# B&R Automation Studio project Kesim (part 3)

#### Park.st
```iecst
ACTION Park:

	CASE gMain.Out.MainSubStep OF

		SUB_INIT:

			IF Loc.FirstInSubState THEN
				gAxBasic[AX_X].MoveAbsolute		:= FALSE;
				gAxBasic[AX_Y].MoveAbsolute		:= FALSE;
				gAxBasic[AX_C].MoveAbsolute		:= FALSE;
				gIO.Out.CT.CuttingHeadDown 		:= FALSE;
				gIO.Out.CT.LowEMotorDown   		:= FALSE;
				gIO.Out.CT.FanStart		   		:= FALSE;
				gIO.Out.CT.XYGlassBreakControl  := FALSE;
				gIO.Out.CT.TransferBelt			:= FALSE;
				gIO.Out.CT.SquareForward		:= FALSE;
			ELSE
				Loc.Timers.TON_ParkState.IN := TRUE;
				Loc.Timers.TON_ParkState.PT := T#1s;
				IF Loc.Timers.TON_ParkState.Q THEN
					Loc.Timers.TON_ParkState.IN := FALSE;
					gMain.Out.MainSubStep			:= PARK_CHECK_IO;
				END_IF
			END_IF;

		PARK_CHECK_IO:
			IF NOT gIO.In.CT.HeadMaxDownSensor THEN
				gMain.Out.Error 	:= TRUE;
				gMain.Out.ErrorID 	:= 999; // Diamond Is Not Back
				gMain.Out.MainSubStep   	:= SUB_ERROR;
				RETURN;

			ELSIF gParameters.MachineType = OCKM THEN
				IF NOT gIO.In.CT.TableDownStopSwicth OR gIO.In.CT.TableUpSlowSwicth ELSE
					gMain.Out.Error 	:= TRUE;
					gMain.Out.ErrorID 	:= 999; // CT_Is_Not_Down
					gMain.Out.MainSubStep   	:= PARK_ERROR;
					RETURN;
					ELSIF NOT gIO.In.CT.TableSquareBack THEN
					gMain.Out.Error 	:= TRUE;
					gMain.Out.ErrorID 	:= 999; // CT_Is_Squares_Are_Not_Back
					gMain.Out.MainSubStep   	:= PARK_ERROR;
					RETURN;
				ELSE
					gMain.Out.MainSubStep   	:= SUB_PARK_START;
				END_IF // OCKM
			ELSIF gParameters.MachineType = FCL THEN
				IF NOT gIO.In.CT.GlassTransBeltIsDown ELSE
					gMain.Out.Error 	:= TRUE;
					gMain.Out.ErrorID 	:= 999; // CT_Belt Is Not Down
					gMain.Out.MainSubStep   	:= SUB_ERROR;
					RETURN;
				END_IF // FCL
			ELSE
				gMain.Out.MainSubStep := SUB_PARK_START;
			END_IF;

			SUB_PARK_START:
				IF Loc.FirstInSubState THEN

					// X Axis Go Park
					gAxBasicPar[AX_X].Acceleration	:= 200.0;
					gAxBasicPar[AX_X].Deceleration 	:= 200.0;
					gAxBasicPar[AX_X].Velocity		:= (gParameters.LengthParametes.ParkSpeed / 100) * C_MAX_CUT_SPEED * (1000/60);
					gAxBasicPar[AX_X].Position 		:= gMain.In.Settings.ParkPos[AX_X];
					gAxBasic[AX_X].MoveAbsolute		:= TRUE;

					// Y Axis Go Park
					gAxBasicPar[AX_Y].Acceleration	:= 200.0;
					gAxBasicPar[AX_Y].Deceleration 	:= 200.0;
					gAxBasicPar[AX_Y].Velocity		:= (gParameters.LengthParametes.ParkSpeed / 100) * C_MAX_CUT_SPEED * (1000/60);
					gAxBasicPar[AX_Y].Position 		:= gMain.In.Settings.ParkPos[AX_Y];
					gAxBasic[AX_Y].MoveAbsolute		:= TRUE;

					// C Axis Go Park
					gAxBasicPar[AX_C].Acceleration	:= 200.0;
					gAxBasicPar[AX_C].Deceleration 	:= 200.0;
					gAxBasicPar[AX_C].Velocity		:= 200.0;
					gAxBasicPar[AX_C].Position 		:= gMain.In.Settings.ParkPos[AX_C];
					gAxBasic[AX_C].MoveAbsolute		:= TRUE;

				ELSE
					IF gAxBasic[AX_X].MoveDone AND gAxBasic[AX_Y].MoveDone AND gAxBasic[AX_C].MoveDone THEN
						gMain.Out.MainSubStep			:= PARK_DONE;
					END_IF;
				END_IF;

			SUB_CMD_DONE:
				IF gMain.Out.Status.Ax_Parked  THEN
					Loc.HomeState			:= SUB_INIT;
					//		gMain.Out.MainStep		:= MAIN_WAIT_CMD;
				END_IF;

			SUB_STOP:

			SUB_ERROR:
			IF Loc.FirstInSubState THEN
				gAxBasic[AX_X].MoveAbsolute		:= FALSE;
				gAxBasic[AX_Y].MoveAbsolute		:= FALSE;
				gAxBasic[AX_C].MoveAbsolute		:= FALSE;
				Loc.Timers.TON_ParkState.IN		:= FALSE;
			ELSE
				IF gMain.In.Cmd.Reset THEN
					gAxBasic[AX_X].ErrorReset		:= TRUE;
					gAxBasic[AX_Y].ErrorReset		:= TRUE;
					gAxBasic[AX_C].ErrorReset		:= TRUE;
				ELSE
					gAxBasic[AX_X].ErrorReset		:= FALSE;
					gAxBasic[AX_Y].ErrorReset		:= FALSE;
					gAxBasic[AX_C].ErrorReset		:= FALSE;
				END_IF;

				IF NOT gAxBasic[ AX_X].Error AND NOT gAxBasic[ AX_Y].Error NOT gAxBasic[ AX_C].Error THEN
					gMain.Out.MainSubStep			:= SUB_INIT;
					//gMain.Out.MainStep		:= MAIN_WAIT_CMD;
				END_IF;

			END_IF;

		END_CASE;

		Loc.Timers.TON_ParkState();

		END_ACTION
```

### Program Logical/SourceCode/CncCtrl (IEC)

#### Main.st - Init, cyclic, exit code
```iecst
(********************************************************************
 * COPYRIGHT --  B&R Industrial Automation GmbH
 ********************************************************************
 * Task: SUB0
 * Author: kay3a
 * Created: October 16, 2024/11:06 AM
 ********************************************************************
 * Description: Machine CncCtrl task
 ********************************************************************)
PROGRAM _INIT

	//|ŻŻŻŻŻŻŻŻŻŻŻŻŻŻŻŻŻŻŻŻŻŻŻŻŻŻŻŻŻŻŻŻŻŻŻŻŻŻŻŻŻŻŻŻŻŻŻŻŻŻŻŻŻŻŻŻŻŻŻŻŻŻŻŻŻŻŻŻŻŻŻŻŻ
	//|               CNC Klasörünü olustur
	//|_________________________________________________________________________
	Loc.FB.DirCreate.Parameters.DeviceName := 'DEV_CNC';
	Loc.FB.DirCreate.Parameters.DirPath := '/DEVICE=USER_PATH/CNC';
	Loc.FB.DirCreate.Enable := TRUE;
	REPEAT
		Loc.FB.DirCreate.Execute := Loc.FB.DirCreate.Active AND NOT Loc.FB.DirCreate.CommandBusy AND NOT Loc.FB.DirCreate.CommandDone;
		Loc.FB.DirCreate();
		UNTIL Loc.FB.DirCreate.CommandDone
	END_REPEAT;
	//|_________________________________________________________________________

	//|ŻŻŻŻŻŻŻŻŻŻŻŻŻŻŻŻŻŻŻŻŻŻŻŻŻŻŻŻŻŻŻŻŻŻŻŻŻŻŻŻŻŻŻŻŻŻŻŻŻŻŻŻŻŻŻŻŻŻŻŻŻŻŻŻŻŻŻŻŻŻŻŻŻ
	//|               CNC File olustur
	//|_________________________________________________________________________
	Loc.FB.FileCreate.Parameters.DeviceName := 'DEV_CNC';
	Loc.FB.FileCreate.Parameters.FileName := 'Program.cnc';
	Loc.FB.FileCreate.Enable := TRUE;
	REPEAT
		Loc.FB.FileCreate.Execute := Loc.FB.FileCreate.Active AND NOT Loc.FB.FileCreate.CommandBusy AND NOT Loc.FB.FileCreate.CommandDone;
		Loc.FB.FileCreate();
		UNTIL Loc.FB.FileCreate.CommandDone
	END_REPEAT;
	//|_________________________________________________________________________

	//|ŻŻŻŻŻŻŻŻŻŻŻŻŻŻŻŻŻŻŻŻŻŻŻŻŻŻŻŻŻŻŻŻŻŻŻŻŻŻŻŻŻŻŻŻŻŻŻŻŻŻŻŻŻŻŻŻŻŻŻŻŻŻŻŻŻŻŻŻŻŻŻŻŻ
	//|               L I V E    F B s
	//|_________________________________________________________________________
//	(* PML *)
//	Loc.FB.PML.MpLink := ADR(gMpLink_PackMLSyncModule_CncCtrl);
//	Loc.FB.PML.Parameters := ADR(Loc.Par.PML);
//	Loc.FB.PML.Enable := TRUE;

	(* CNC *)
	Loc.FB.Cnc3Axis.MpLink := ADR(gMpLink_CncXYZ);
	Loc.FB.Cnc3Axis.Parameters := ADR(Loc.Par.Cnc3Axis);
	Loc.FB.Cnc3Axis.Enable := TRUE;
	Loc.FB.Cnc3Axis.Override := 100.0;
	// Par
	Loc.Par.Cnc3Axis.ProgramName := 'Program.cnc';
	//|_________________________________________________________________________

END_PROGRAM

PROGRAM _CYCLIC

	(* Axis *)
	Loc.FB.Cnc3Axis();

	//|_________________________________________________________________________
	TestX := Loc.FB.Cnc3Axis.X / 1500;
	TestY := Loc.FB.Cnc3Axis.Z / 1500;

  gCncAdress := ADR ( Loc.FB.Cnc3Axis );

END_PROGRAM

PROGRAM _EXIT

	//|ŻŻŻŻŻŻŻŻŻŻŻŻŻŻŻŻŻŻŻŻŻŻŻŻŻŻŻŻŻŻŻŻŻŻŻŻŻŻŻŻŻŻŻŻŻŻŻŻŻŻŻŻŻŻŻŻŻŻŻŻŻŻŻŻŻŻŻŻŻŻŻŻŻ
	//|              K I L L   F B s
	//|_________________________________________________________________________
	(* PML *)
//	Loc.FB.PML(Enable := FALSE);

	(* CNC *)
	Loc.FB.Cnc3Axis(Enable := FALSE);
	//|_________________________________________________________________________

END_PROGRAM
```

#### Types.typ - Local data types
```iecst
(********************************************************************
 * COPYRIGHT --  B&R Industrial Automation GmbH
 *******************************************************************
 * Task: MAIN
 * Author: kay3a
 * Created: October 16, 2024/11:08 AM
 ********************************************************************)

TYPE
	Loc_typ : 	STRUCT  (**** Local Type*)
		FB : Loc_FB_typ; (**** Local FB Type*)
		Par : Loc_Par_typ;
		Cmd : Loc_Cmd_typ; (**** Local Command Type*)
		Status : Loc_Status_typ; (**** Local Status Type*)
	END_STRUCT;
END_TYPE

(**)
(**** Local FB Type*)

TYPE
	Loc_FB_typ : 	STRUCT  (**** Local FB Type*)
		Cnc3Axis : MpCnc3Axis; (**** CNC FB*)
		DirCreate : FbDirCreate; (**** CNC Direction create*)
		FileCreate : FbFileCreate; (**** CNC File create*)
	END_STRUCT;
END_TYPE

(**)
(**** Local Par Type*)

TYPE
	Loc_Par_typ : 	STRUCT  (**** Local Par Type*)
		Cnc3Axis : MpCnc3AxisParType;
	END_STRUCT;
END_TYPE

(**)
(**** Local Cmd Type*)

TYPE
	Loc_Cmd_typ : 	STRUCT  (**** Local Cmd Type*)
		New_Member : USINT;
	END_STRUCT;
END_TYPE

(**)
(**** Local Status Type*)

TYPE
	Loc_Status_typ : 	STRUCT  (**** Local Status Type*)
		New_Member : USINT;
	END_STRUCT;
END_TYPE

(**)
```

#### Variables.var - Local variables
```iecst
(********************************************************************
 * COPYRIGHT --  B&R Industrial Automation GmbH
 *******************************************************************
 * Task: MAIN
 * Author: kay3a
 * Created: October 16, 2024/11:08 AM
 ********************************************************************)
VAR
	Loc : Loc_typ; (**** Bu Task icinde kullanilacak Local degisken*)
	TestY : LREAL;
	TestX : LREAL;
END_VAR
```

#### Package Logical/SourceCode/CncCtrl/act_PML - PackML specific actions are stored in this package.

#### Execute.st
```iecst
(*********************************************************************************
 * Copyright: B&R Industrial Automation GmbH
 * Author:    kay3a
 * Created:   June 21, 2023/5:55 PM
 *********************************************************************************)
ACTION Execute:

END_ACTION

ACTION Execute_Manual:

END_ACTION

ACTION Execute_Production:

END_ACTION
```

#### Starting.st
```iecst
(*********************************************************************************
 * Copyright: B&R Industrial Automation GmbH
 * Author:    kay3a
 * Created:   June 21, 2023/5:55 PM
 *********************************************************************************)
ACTION Starting:

	Loc.FB.PML.Command.StateComplete := TRUE;

END_ACTION
```

#### Stopping.st
```iecst
(*********************************************************************************
 * Copyright: B&R Industrial Automation GmbH
 * Author:    kay3a
 * Created:   June 21, 2023/5:55 PM
 *********************************************************************************)
ACTION Stopping:

Loc.FB.PML.Command.StateComplete := TRUE;

END_ACTION
```

#### Completing.st
```iecst
(*********************************************************************************
 * Copyright: B&R Industrial Automation GmbH
 * Author:    kay3a
 * Created:   June 21, 2023/5:55 PM
 *********************************************************************************)
ACTION Completing:

Loc.FB.PML.Command.StateComplete := TRUE;

END_ACTION
```

#### Suspended.st
```iecst
(*********************************************************************************
 * Copyright: B&R Industrial Automation GmbH
 * Author:    kay3a
 * Created:   June 21, 2023/5:55 PM
 *********************************************************************************)
ACTION Suspended:

Loc.FB.PML.Command.StateComplete := TRUE;

END_ACTION
```

#### Complete.st
```iecst
(*********************************************************************************
 * Copyright: B&R Industrial Automation GmbH
 * Author:    kay3a
 * Created:   June 21, 2023/5:55 PM
 *********************************************************************************)
ACTION Complete:

END_ACTION
```

#### Idle.st
```iecst
(*********************************************************************************
 * Copyright: B&R Industrial Automation GmbH
 * Author:    kay3a
 * Created:   June 21, 2023/5:55 PM
 *********************************************************************************)
ACTION Idle:

END_ACTION
```

#### Unholding.st
```iecst
(*********************************************************************************
 * Copyright: B&R Industrial Automation GmbH
 * Author:    kay3a
 * Created:   June 21, 2023/5:55 PM
 *********************************************************************************)
ACTION Unholding:

	Loc.FB.PML.Command.StateComplete := TRUE;

END_ACTION
```

#### Held.st
```iecst
(*********************************************************************************
 * Copyright: B&R Industrial Automation GmbH
 * Author:    kay3a
 * Created:   June 21, 2023/5:55 PM
 *********************************************************************************)
ACTION Held:

END_ACTION
```

- sample.pptx (binary file, 35832 bytes)
#### GCode_Ref.txt
```
%001 (CncProgram)

N10 G90     (absolute coordinates)
N20 F10000    (Feed rate in measurements units/min)

(* Glass Height:1500mm
(* Glass Length:1000mm  *)

G04 3
G01 X 0  Y0  Z0
G01 X-1000
G01 Y-90
G01 Z1000

G03  G18 I500 H180   Z1000 Y-270

G01 Z0
```

### Program Logical/SourceCode/Infastructure/AlarmX (IEC)

#### Main.st - Init, cyclic, exit code
```iecst
(********************************************************************
 * COPYRIGHT --  B&R Industrial Automation GmbH
 ********************************************************************
 * Task: AlarmX
 * Author: kay3a
 * Created: October 2, 2024/3:55 PM
 ********************************************************************
 * Description: Alarm mgr
 ********************************************************************)
PROGRAM _INIT

	//|ŻŻŻŻŻŻŻŻŻŻŻŻŻŻŻŻŻŻŻŻŻŻŻŻŻŻŻŻŻŻŻŻŻŻŻŻŻŻŻŻŻŻŻŻŻŻŻŻŻŻŻŻŻŻŻŻŻŻŻŻŻŻŻŻŻŻŻŻŻŻŻŻŻ
	//|               AlarmXHistory Klasörünü olustur
	//|_________________________________________________________________________
	Loc.FB.DirCreate.Parameters.DeviceName := 'DEV_ALARM';
	Loc.FB.DirCreate.Parameters.DirPath := '/DEVICE=USER_PATH/AlarmX';
	Loc.FB.DirCreate.Enable := TRUE;
	REPEAT
		Loc.FB.DirCreate.Execute := Loc.FB.DirCreate.Active AND NOT Loc.FB.DirCreate.CommandBusy AND NOT Loc.FB.DirCreate.CommandDone;
		Loc.FB.DirCreate();
		UNTIL Loc.FB.DirCreate.CommandDone
	END_REPEAT;
	//|_________________________________________________________________________

	//|ŻŻŻŻŻŻŻŻŻŻŻŻŻŻŻŻŻŻŻŻŻŻŻŻŻŻŻŻŻŻŻŻŻŻŻŻŻŻŻŻŻŻŻŻŻŻŻŻŻŻŻŻŻŻŻŻŻŻŻŻŻŻŻŻŻŻŻŻŻŻŻŻŻ
	//|               FB linklemeleri
	//|_________________________________________________________________________
	(* AlarmXCore *)
	Loc.FB.AlarmXCore.MpLink := ADR(gMpLink_AlarmXCore);
	Loc.FB.AlarmXCore.Enable := TRUE;
	Loc.FB.AlarmXCore();

	(* AlarmXHistory *)
	Loc.FB.AlarmXHistory.Enable := TRUE;
	Loc.FB.AlarmXHistory.MpLink := ADR(gMpLink_AlarmXHistory);
	Loc.FB.AlarmXHistory.FileName := ADR('Alarms_%Y_%m_%d_%H_%M_%S');
	Loc.FB.AlarmXHistory.DeviceName := ADR('DEV_ALARM');
	Loc.FB.AlarmXHistory();
	//|_________________________________________________________________________

	//|ŻŻŻŻŻŻŻŻŻŻŻŻŻŻŻŻŻŻŻŻŻŻŻŻŻŻŻŻŻŻŻŻŻŻŻŻŻŻŻŻŻŻŻŻŻŻŻŻŻŻŻŻŻŻŻŻŻŻŻŻŻŻŻŻŻŻŻŻŻŻŻŻŻ
	//|               Ilk Açilis AlarmHist temizle
	//|_________________________________________________________________________
//	Loc.FB.AlarmXHistory.Clear := TRUE; // bc25.10.15
	//|_________________________________________________________________________

END_PROGRAM

PROGRAM _CYCLIC

	//|ŻŻŻŻŻŻŻŻŻŻŻŻŻŻŻŻŻŻŻŻŻŻŻŻŻŻŻŻŻŻŻŻŻŻŻŻŻŻŻŻŻŻŻŻŻŻŻŻŻŻŻŻŻŻŻŻŻŻŻŻŻŻŻŻŻŻŻŻŻŻŻŻŻ
	//|                Command set/reset
	//|_________________________________________________________________________
	(* AlarmXHistory FB --- ErrorReset *)
	IF Loc.FB.AlarmXHistory.Error THEN
		Loc.FB.AlarmXHistory.ErrorReset := TRUE;
	ELSE
		Loc.FB.AlarmXHistory.ErrorReset := FALSE;
	END_IF;

	(* AlarmXCore FB --- ErrorReset *)
	IF Loc.FB.AlarmXCore.Error THEN
		Loc.FB.AlarmXCore.ErrorReset := TRUE;
	ELSE
		Loc.FB.AlarmXCore.ErrorReset := FALSE;
	END_IF;

	(* AlarmXCore --- AcknowledgeAll *)
	IF Loc.FB.AlarmXCore.CommandDone THEN
		Loc.FB.AlarmXCore.AcknowledgeAll := FALSE;
	ELSE
		IF Loc.Cmd.AcknowledgeAll AND Loc.FB.AlarmXCore.UnacknowledgedAlarms <> 0 THEN
			Loc.FB.AlarmXCore.AcknowledgeAll := TRUE;
		END_IF;
	END_IF;
	//|_________________________________________________________________________

	//|ŻŻŻŻŻŻŻŻŻŻŻŻŻŻŻŻŻŻŻŻŻŻŻŻŻŻŻŻŻŻŻŻŻŻŻŻŻŻŻŻŻŻŻŻŻŻŻŻŻŻŻŻŻŻŻŻŻŻŻŻŻŻŻŻŻŻŻŻŻŻŻŻŻ
	//|               AlarmX Category check
	//|_________________________________________________________________________
	// Category isimlerinin Category.Cfg tablosundaki ile ayni olmasi gerekmekte
	Loc.Status.ReactionCategory[LC_ALARM_Category0_Abort] := MpAlarmXCheckReaction(gMpLink_AlarmXCore, 'Category0_Abort');
	Loc.Status.ReactionCategory[LC_ALARM_Category1_Stop]  := MpAlarmXCheckReaction(gMpLink_AlarmXCore, 'Category1_Stop');
	Loc.Status.ReactionCategory[LC_ALARM_Category2_Pause] := MpAlarmXCheckReaction(gMpLink_AlarmXCore, 'Category2_Pause');
	Loc.Status.ReactionCategory[LC_ALARM_Category3_Info]  := MpAlarmXCheckReaction(gMpLink_AlarmXCore, 'Category3_Info');
	//|_________________________________________________________________________

	//|ŻŻŻŻŻŻŻŻŻŻŻŻŻŻŻŻŻŻŻŻŻŻŻŻŻŻŻŻŻŻŻŻŻŻŻŻŻŻŻŻŻŻŻŻŻŻŻŻŻŻŻŻŻŻŻŻŻŻŻŻŻŻŻŻŻŻŻŻŻŻŻŻŻ
	//|              Helper Actions
	//|_________________________________________________________________________
	Interaction;
	AutoExport;
	AlarmHandle;
	//|_________________________________________________________________________

	//|ŻŻŻŻŻŻŻŻŻŻŻŻŻŻŻŻŻŻŻŻŻŻŻŻŻŻŻŻŻŻŻŻŻŻŻŻŻŻŻŻŻŻŻŻŻŻŻŻŻŻŻŻŻŻŻŻŻŻŻŻŻŻŻŻŻŻŻŻŻŻŻŻŻ
	//|               FB Call
	//|_________________________________________________________________________
	Loc.FB.AlarmXCore();
	Loc.FB.AlarmXHistory();
	//|_________________________________________________________________________

	gHMI.CommUnit.ActAlarms := Loc.FB.AlarmXCore.PendingAlarms;
END_PROGRAM

PROGRAM _EXIT

	//|ŻŻŻŻŻŻŻŻŻŻŻŻŻŻŻŻŻŻŻŻŻŻŻŻŻŻŻŻŻŻŻŻŻŻŻŻŻŻŻŻŻŻŻŻŻŻŻŻŻŻŻŻŻŻŻŻŻŻŻŻŻŻŻŻŻŻŻŻŻŻŻŻŻ
	//|               FB Kill
	//|_________________________________________________________________________
	Loc.FB.AlarmXCore(Enable := FALSE);
	Loc.FB.AlarmXHistory(Enable := FALSE);
	//|_________________________________________________________________________

END_PROGRAM
```

#### Types.typ - Local data types
```iecst
(********************************************************************
 * COPYRIGHT --  B&R Industrial Automation GmbH
 *******************************************************************
 * Task: AlarmX
 * Author: kay3a
 * Created: October 2, 2024/3:56 PM
 ********************************************************************)
(**)
(**** Local Type*)

TYPE
	Loc_typ : 	STRUCT  (**** Local Type*)
		FB : Loc_FB_typ; (**** Local FB Type*)
		Cmd : Loc_Cmd_typ; (**** Local Command Type*)
		Status : Loc_Status_typ; (**** Local Status Type*)
	END_STRUCT;
END_TYPE

(**)
(**** Local FB Type*)

TYPE
	Loc_FB_typ : 	STRUCT  (**** Local FB Type*)
		DirCreate : FbDirCreate; (**** Alarm geçmisi export dosyalarini tutmak için*)
		AlarmXCore : MpAlarmXCore; (**** Local FB AlarmXCore Type*)
		AlarmXHistory : MpAlarmXHistory; (**** Local FB AlarmXHistory Type*)
	END_STRUCT;
END_TYPE

(**)
(**** Local Cmd Type*)

TYPE
	Loc_Cmd_typ : 	STRUCT  (**** Local Cmd Type*)
		AcknowledgeAll : BOOL; (**** Tüm alarmlari onayla*)
		AutoExport : BOOL; (**** Alarm geçmisini export et.*)
	END_STRUCT;
END_TYPE

(**)
(**** Local Status Type*)

TYPE
	Loc_Status_typ : 	STRUCT  (**** Local Status Type*)
		Alerts : Loc_Status_Alerts_typ; (**** Alarm durumlari*)
		ReactionCategory : ARRAY[0..LC_MAX_ALARM_CATEGORY_INDEX]OF BOOL; (**** Alarm reaction durumlari.*)
	END_STRUCT;
END_TYPE

(**)
(**** Local Status Alarm Type*)

TYPE
	Loc_Status_Alerts_typ : 	STRUCT  (**** Local Status Alarm Type*)
		Single : Loc_Status_Alerts_Single_typ; (**** Single alarm durumlari*)
		Snippet : ARRAY[0..LC_MAX_SNIPPET_ALARM_INDEX]OF Loc_Status_Alerts_Snippet_typ; (**** Snppet alarm durumlari ve index leri*)
	END_STRUCT;
END_TYPE

(**)
(**** Local Status Alarm Single Type*)

TYPE
	Loc_Status_Alerts_Single_typ : 	STRUCT  (**** Local Status Alarm Single Type*)
		Abort : ARRAY[0..MAX_SINGLE_ALARM_MIN1]OF BOOL;
		Stop : ARRAY[0..MAX_SINGLE_ALARM_MIN1]OF BOOL;
		Pause : ARRAY[0..MAX_SINGLE_ALARM_MIN1]OF BOOL;
		Info : ARRAY[0..MAX_SINGLE_ALARM_MIN1]OF BOOL;
	END_STRUCT;
END_TYPE

(**)
(**** Local Status Alarm Snippet Type*)

TYPE
	Loc_Status_Alerts_Snippet_typ : 	STRUCT  (**** Local Status Alarm Snippet Type*)
		Index : DINT; (**** Snippet alarm index degeri*)
		Val : BOOL; (**** Snippet alarm degeri*)
	END_STRUCT;
END_TYPE

(**)
```

#### AlarmHandle.st
```iecst
(********************************************************************
 * COPYRIGHT --  B&R Industrial Automation GmbH
 ********************************************************************
 * Task: AlarmX
 * Author: kay3a
 * Created: October 2, 2024/11:08 PM
 ********************************************************************
 * Description: Alarms Handle action.
 ********************************************************************)
//==============================================================================
ACTION AlarmHandle:

	//|ŻŻŻŻŻŻŻŻŻŻŻŻŻŻŻŻŻŻŻŻŻŻŻŻŻŻŻŻŻŻŻŻŻŻŻŻŻŻŻŻŻŻŻŻŻŻŻŻŻŻŻŻŻŻŻŻŻŻŻŻŻŻŻŻŻŻŻŻŻŻŻŻŻ
	//|               Read Global Alerts
	//|_________________________________________________________________________
	brsmemcpy(ADR(Loc.Status.Alerts.Single.Abort), ADR(gAlert.Abort.IDX), SIZEOF(Loc.Status.Alerts.Single.Abort));
	brsmemcpy(ADR(Loc.Status.Alerts.Single.Stop),  ADR(gAlert.Stop.IDX),  SIZEOF(Loc.Status.Alerts.Single.Stop));
	brsmemcpy(ADR(Loc.Status.Alerts.Single.Pause), ADR(gAlert.Pause.IDX), SIZEOF(Loc.Status.Alerts.Single.Pause));
	brsmemcpy(ADR(Loc.Status.Alerts.Single.Info),  ADR(gAlert.Info.IDX),  SIZEOF(Loc.Status.Alerts.Single.Info));
	//|_________________________________________________________________________

	//|ŻŻŻŻŻŻŻŻŻŻŻŻŻŻŻŻŻŻŻŻŻŻŻŻŻŻŻŻŻŻŻŻŻŻŻŻŻŻŻŻŻŻŻŻŻŻŻŻŻŻŻŻŻŻŻŻŻŻŻŻŻŻŻŻŻŻŻŻŻŻŻŻŻ
	//|               	Clear Global Alarm ID
	//|_________________________________________________________________________
	brsmemset(ADR(gAlert.Abort.IDX), 0, SIZEOF(gAlert.Abort.IDX));
	brsmemset(ADR(gAlert.Stop.IDX),  0, SIZEOF(gAlert.Stop.IDX));
	brsmemset(ADR(gAlert.Pause.IDX), 0, SIZEOF(gAlert.Pause.IDX));
	brsmemset(ADR(gAlert.Info.IDX),  0, SIZEOF(gAlert.Info.IDX));
	//|_________________________________________________________________________

END_ACTION
//==============================================================================

//==============================================================================
ACTION SnippetAlerts:

	//|ŻŻŻŻŻŻŻŻŻŻŻŻŻŻŻŻŻŻŻŻŻŻŻŻŻŻŻŻŻŻŻŻŻŻŻŻŻŻŻŻŻŻŻŻŻŻŻŻŻŻŻŻŻŻŻŻŻŻŻŻŻŻŻŻŻŻŻŻŻŻŻŻŻ
	//|               Snippet alarms genarate
	//|_________________________________________________________________________
	Loc.Status.Alerts.Snippet[0].Index;
	Loc.Status.Alerts.Snippet[0].Val;

	Loc.Status.Alerts.Snippet[1].Index;
	Loc.Status.Alerts.Snippet[1].Val;

	Loc.Status.Alerts.Snippet[2].Index;
	Loc.Status.Alerts.Snippet[2].Val;

	Loc.Status.Alerts.Snippet[3].Index;
	Loc.Status.Alerts.Snippet[3].Val;

	Loc.Status.Alerts.Snippet[4].Index;
	Loc.Status.Alerts.Snippet[4].Val;

	Loc.Status.Alerts.Snippet[5].Index;
	Loc.Status.Alerts.Snippet[5].Val;

	Loc.Status.Alerts.Snippet[6].Index;
	Loc.Status.Alerts.Snippet[6].Val;

	Loc.Status.Alerts.Snippet[7].Index;
	Loc.Status.Alerts.Snippet[7].Val;

	Loc.Status.Alerts.Snippet[8].Index;
	Loc.Status.Alerts.Snippet[8].Val;

	Loc.Status.Alerts.Snippet[9].Index;
	Loc.Status.Alerts.Snippet[9].Val;

	Loc.Status.Alerts.Snippet[10].Index;
	Loc.Status.Alerts.Snippet[10].Val;
	//|_________________________________________________________________________

END_ACTION
//==============================================================================
```

#### Interaction.st
```iecst
(********************************************************************
 * COPYRIGHT --  B&R Industrial Automation GmbH
 ********************************************************************
 * Task: AlarmX
 * Author: kay3a
 * Created: October 3, 2024/10:48 AM
 ********************************************************************
 * Description: Local/ global degiskenler arasinda okuma yazma yapar.
 ********************************************************************)
//==============================================================================
ACTION Interaction:

	//|ŻŻŻŻŻŻŻŻŻŻŻŻŻŻŻŻŻŻŻŻŻŻŻŻŻŻŻŻŻŻŻŻŻŻŻŻŻŻŻŻŻŻŻŻŻŻŻŻŻŻŻŻŻŻŻŻŻŻŻŻŻŻŻŻŻŻŻŻŻŻŻŻŻ
	//|               Local / Global variables     ---   READ / WRITE
	//|_________________________________________________________________________
	(* READ from Global *)
//	Loc.Cmd.AcknowledgeAll := gCommUnit.Main.In.MachineReset;
//
//

	(* WRTIE to Global *)
	gAlert.Abort.Status := Loc.Status.ReactionCategory[LC_ALARM_Category0_Abort];
	gAlert.Stop.Status  := Loc.Status.ReactionCategory[LC_ALARM_Category1_Stop];
	gAlert.Pause.Status := Loc.Status.ReactionCategory[LC_ALARM_Category2_Pause];
	gAlert.Info.Status	:= Loc.Status.ReactionCategory[LC_ALARM_Category3_Info];
	//|_________________________________________________________________________

END_ACTION
//==============================================================================
```

#### AutoExport.st
```iecst
(********************************************************************
 * COPYRIGHT --  B&R Industrial Automation GmbH
 ********************************************************************
 * Task: AlarmX
 * Author: kay3a
 * Created: October 3, 2024/2:53 PM
 ********************************************************************
 * Description: Belirlenen kosullar sonrasinda AutoExport komutu olusturur.
 ********************************************************************)
ACTION AutoExport:

	//|ŻŻŻŻŻŻŻŻŻŻŻŻŻŻŻŻŻŻŻŻŻŻŻŻŻŻŻŻŻŻŻŻŻŻŻŻŻŻŻŻŻŻŻŻŻŻŻŻŻŻŻŻŻŻŻŻŻŻŻŻŻŻŻŻŻŻŻŻŻŻŻŻŻ
	//|               AutoExport Genarate
	//|_________________________________________________________________________
	// belirli tarihlerde veya belirli sayiya ulasildiginda Auto Export yapilabilir.
	Loc.Cmd.AutoExport;
	//|_________________________________________________________________________

END_ACTION
```

### Program Logical/SourceCode/Infastructure/UserXMgr (IEC)

#### Main.st - Init, cyclic, exit code
```iecst
(********************************************************************
* COPYRIGHT --  B&R Industrial Automation GmbH
********************************************************************
* Task: UserX
* Author: kay3a
* Created: October 3, 2024/4:57 PM
********************************************************************
* Description: UserX manager
********************************************************************)
PROGRAM _INIT

//|ŻŻŻŻŻŻŻŻŻŻŻŻŻŻŻŻŻŻŻŻŻŻŻŻŻŻŻŻŻŻŻŻŻŻŻŻŻŻŻŻŻŻŻŻŻŻŻŻŻŻŻŻŻŻŻŻŻŻŻŻŻŻŻŻŻŻŻŻŻŻŻŻŻ
//|               UserX Klasörünü olustur
//|_________________________________________________________________________
	Loc.FB.DirCreate.Parameters.DeviceName := 'DEV_USER';
	Loc.FB.DirCreate.Parameters.DirPath := '/DEVICE=USER_PATH/UserX';
	Loc.FB.DirCreate.Enable := TRUE;
	REPEAT
		Loc.FB.DirCreate.Execute := Loc.FB.DirCreate.Active AND NOT Loc.FB.DirCreate.CommandBusy AND NOT Loc.FB.DirCreate.CommandDone;
		Loc.FB.DirCreate();
		UNTIL Loc.FB.DirCreate.CommandDone
	END_REPEAT;
	//|_________________________________________________________________________

	//|ŻŻŻŻŻŻŻŻŻŻŻŻŻŻŻŻŻŻŻŻŻŻŻŻŻŻŻŻŻŻŻŻŻŻŻŻŻŻŻŻŻŻŻŻŻŻŻŻŻŻŻŻŻŻŻŻŻŻŻŻŻŻŻŻŻŻŻŻŻŻŻŻŻ
	//|               FB linklemeleri
	//|_________________________________________________________________________
	(* UserXLogin *)
	Loc.FB.UserXLogin.MpLink := ADR(gMpLink_UserXLogin);
	Loc.FB.UserXLogin.Enable := TRUE;
	Loc.FB.UserXLogin();

	(* UserXLoginUI *)
	Loc.FB.UserXLoginUI.MpLink := ADR(gMpLink_UserXLogin);
	Loc.FB.UserXLoginUI.UIConnect := ADR(Loc.Par.UserXLoginUIConnect);
	Loc.FB.UserXLoginUI.Enable := TRUE;
	Loc.FB.UserXLoginUI();

	(* UserXManagerUI *)
	Loc.Par.UserXMgrUIConnect.User.Create.Lock := FALSE;
	Loc.Par.UserXMgrUIConnect.User.Lock := FALSE;
	Loc.Par.UserXMgrUIConnect.User.Edit.Lock := FALSE;
	Loc.Par.UserXMgrUIConnect.User.Create.Dialog.UserName := "";
	Loc.Par.UserXMgrUIConnect.User.Create.Dialog.NewPassword := "";
	Loc.Par.UserXMgrUIConnect.User.Create.Dialog.ConfirmPassword := "";
	Loc.Par.UserXMgrUIConnect.User.List.MaxSelection := USER_LIST_MAX_SELECTION;
	Loc.Par.UserXMgrUIConnect.User.List.RangeStart := USER_LIST_RANGE_START;
	Loc.Par.UserXMgrUIConnect.User.List.RangeEnd := USER_LIST_RANGE_END;
	Loc.FB.UserXManagerUI.MpLink := ADR(gMpLink_UserXLogin);
	Loc.FB.UserXManagerUI.UIConnect := ADR(Loc.Par.UserXMgrUIConnect);
	Loc.FB.UserXManagerUI.UISetup.FileDevice := 'DEV_USER';
	Loc.FB.UserXManagerUI.Enable := TRUE;
	Loc.FB.UserXManagerUI();
	//|_________________________________________________________________________

END_PROGRAM

PROGRAM _CYCLIC

//|ŻŻŻŻŻŻŻŻŻŻŻŻŻŻŻŻŻŻŻŻŻŻŻŻŻŻŻŻŻŻŻŻŻŻŻŻŻŻŻŻŻŻŻŻŻŻŻŻŻŻŻŻŻŻŻŻŻŻŻŻŻŻŻŻŻŻŻŻŻŻŻŻŻ
//|               Helper Actions
//|_________________________________________________________________________
	HMIAction;
	//|_________________________________________________________________________

	//|ŻŻŻŻŻŻŻŻŻŻŻŻŻŻŻŻŻŻŻŻŻŻŻŻŻŻŻŻŻŻŻŻŻŻŻŻŻŻŻŻŻŻŻŻŻŻŻŻŻŻŻŻŻŻŻŻŻŻŻŻŻŻŻŻŻŻŻŻŻŻŻŻŻ
	//|               Assign
	//|_________________________________________________________________________
	// Saving last status of UserXMgrUIconnect
	Loc.Status.LastMgrConnectStatus := Loc.Par.UserXMgrUIConnect.Status;
	//|_________________________________________________________________________

	//|ŻŻŻŻŻŻŻŻŻŻŻŻŻŻŻŻŻŻŻŻŻŻŻŻŻŻŻŻŻŻŻŻŻŻŻŻŻŻŻŻŻŻŻŻŻŻŻŻŻŻŻŻŻŻŻŻŻŻŻŻŻŻŻŻŻŻŻŻŻŻŻŻŻ
	//|               FB Call
	//|_________________________________________________________________________
	Loc.FB.UserXLogin();
	Loc.FB.UserXLoginUI();
	Loc.FB.UserXManagerUI();
	//|_________________________________________________________________________

END_PROGRAM

PROGRAM _EXIT

//|ŻŻŻŻŻŻŻŻŻŻŻŻŻŻŻŻŻŻŻŻŻŻŻŻŻŻŻŻŻŻŻŻŻŻŻŻŻŻŻŻŻŻŻŻŻŻŻŻŻŻŻŻŻŻŻŻŻŻŻŻŻŻŻŻŻŻŻŻŻŻŻŻŻ
//|               FB Kill
//|_________________________________________________________________________
	Loc.FB.UserXLogin(Enable := FALSE);
	Loc.FB.UserXLoginUI(Enable := FALSE);
	Loc.FB.UserXManagerUI(Enable := FALSE);
	//|_________________________________________________________________________

END_PROGRAM
```

#### Variables.var - Local variables
```iecst
(********************************************************************
 * COPYRIGHT --  B&R Industrial Automation GmbH
 *******************************************************************
 * Task: UserX
 * Author: kay3a
 * Created: October 3, 2024/4:59 PM
 ********************************************************************)
(**)
(**** Local variables*)
VAR
	Loc : Loc_typ; (**** Bu Task icinde kullanilacak Local degisken*)
END_VAR
(**)
(**)
(**)
(*Temp Variables*)
VAR
	temp : STRING[255]; (*Temporary string holder for checking file names*)
	i : USINT; (*Index*)
END_VAR
```

### ForcePackage.var
```iecst
(********************************************************************
 * COPYRIGHT -- Bernecker + Rainer
 ********************************************************************
 * Package: ForceIOs
 * File: ForcePackage.var
 * Author: abdullahoglf
 * Created: February 12, 2014
 ********************************************************************
 * Variables of package ForceIOs
 ********************************************************************)
(**)
(**********************************************************************)
(*IO Handling Package Variables*)
(**********************************************************************)
(*State Definitions*)
VAR
	state : USINT := 0;
END_VAR
VAR CONSTANT
	ERROR : USINT := 60;
	GET_LIST : USINT := 55;
	GET_NUM_INFO : USINT := 50;
	DISPOSE_INFO : USINT := 40;
	CREATE_INFO : USINT := 30;
	GET_STR_INFO : USINT := 20;
	MAIN : USINT := 10;
	WAIT_START : USINT := 0;
END_VAR
(*Input Controls*)
VAR
	MyDiagDisposeInfo : DiagDisposeInfo;
	MyDiagCreateInfo : DiagCreateInfo;
	MyDiagGetNumInfo : DiagGetNumInfo;
	MyDiagGetStrInfo : DiagGetStrInfo;
END_VAR
(*Information about the object*)
VAR
	Info : Info_typ;
END_VAR
(*DiagGetNumInfo()*)
VAR
	GetNumInfoCommand : GetNumInfoCommands_typ;
END_VAR
(*DiagGetStrInfo()*)
VAR
	GetStrInfoCommand : GetStrInfoCommands_typ;
END_VAR
(*DiagCreateInfo()*)
VAR
	CreateInfoCommand : CreateInfoCommands_typ;
END_VAR
(*DiagDisposeInfo()*)
VAR
	DisposeInfoCommand : DisposeInfoCommands_typ;
END_VAR
(*Get List*)
VAR
	GetList : GetList_typ;
END_VAR
(*IO Cards Order Check*)
VAR
	ioCfgStart : UDINT := 0; (*Internal index where the storage of IO Card starts in the PLC memory*)
	aiCount : UDINT;
	aiStartIndex : UDINT;
	aoCount : UDINT;
	aoStartIndex : UDINT;
	diCount : UDINT;
	diStartIndex : UDINT;
	doCount : UDINT;
	doStartIndex : UDINT;
END_VAR
(****************************************************************************)
```

### ForcePackage.typ
```iecst
(********************************************************************
 * COPYRIGHT -- Bernecker + Rainer
 ********************************************************************
 * Package: ForceIOs
 * File: ForcePackage.typ
 * Author: abdullahoglf
 * Created: February 12, 2014
 ********************************************************************
 * Data types of package ForceIOs
 ********************************************************************)
(**)
(**************************************************************************************)
(*IO Handling Package Datatypes*)
(**************************************************************************************)

TYPE
	DisposeInfoCommands_typ : 	STRUCT
		disponseInfo : BOOL; (*Cmd to dispose info*)
	END_STRUCT;
END_TYPE

(*I/O's for DiagGetStrInfo()*)

TYPE
	GetStrInfoCommands_typ : 	STRUCT
		infoCode : UDINT; (*Information code configured for the FB*)
		desiredStr : STRING[80]; (*Returned information from the FB*)
		index : UDINT; (*Index of the HW module -- corresponds to an internal order; does not have to be the same with the physical order*)
		getStrInfo : BOOL; (*Cmd to get the information*)
	END_STRUCT;
END_TYPE

(*I/O's for DiagGetStrInfo()*)

TYPE
	GetNumInfoCommands_typ : 	STRUCT
		infoCode : UDINT; (*Information code configured for the FB*)
		index : UDINT; (*Index of the HW module -- corresponds to an internal order; does not have to be the same with the physical order*)
		getNumInfo : BOOL; (*Cmd to get the numeric information*)
		desiredNum : UDINT; (*Returned numric info from the FB*)
	END_STRUCT;
END_TYPE

(*I/O's for DiagCreateInfo()*)

TYPE
	CreateInfoCommands_typ : 	STRUCT
		plugged : BOOL; (*Cmd to get information about the plugged HW modules*)
		createInfo : BOOL; (*Cmd to get the information*)
		configured : BOOL; (*Cmd to get information about the configured HW modules*)
		all : BOOL; (*Cmd to get information about all the HW modules*)
	END_STRUCT;
	Info_typ : 	STRUCT
		NumbersEntries : UDINT; (*Number of entries*)
		Ident : UDINT; (*ID of the information *)
		errorAck : BOOL; (*Error acknowledgement button*)
		errorFlag : BOOL; (*Error flag*)
		errorStatement : STRING[80]; (*Error statement*)
		Index : UDINT; (*Index for the list*)
	END_STRUCT;
END_TYPE

(*Default values for the list*)

TYPE
	List_typ : 	STRUCT
		moduleState : UDINT; (*Module state --- 1 = configured but not plugged; 2 = inserted but not configured; 3 = configured & plugged; 4 = inserted module is different than the configured module*)
		name : STRING[80]; (*Returned HW module name*)
		index : UDINT; (*Index of the HW module -- corresponds to an internal order; does not have to be the same with the physical order*)
	END_STRUCT;
END_TYPE

(*I/O's for GET_LIST*)

TYPE
	GetList_typ : 	STRUCT
		List : ARRAY[0..100]OF List_typ; (*The HW module information list*)
		GetList : BOOL; (*Cmd to create the list*)
	END_STRUCT;
END_TYPE
```

### Program Logical/SourceCode/Infastructure/ForceIOs/ForceIO (IEC)

#### Main.st - Init, cyclic, exit code
```iecst
(********************************************************************
 * COPYRIGHT -- Bernecker + Rainer
 ********************************************************************
 * PROGRAM: ForceIO
 * File: ForceIO.st
 * Author: abdullahoglf
 * Created: December 18, 2013
 ********************************************************************
 * Implementation OF PROGRAM ForceIO
 ********************************************************************)

PROGRAM _INIT

	forceStep   := FORCE_WAIT;

	// run GetSignalStr once so that GetDPStatus has a valid datapoint to start with
	GetSignalStr_1.uNumStation    := slotIndex + 1;    // configured for GetSignalStr
	GetSignalStr_1.uNumSignal     := j + 1;		    // configured for GetSignalStr
	GetSignalStr_0.uNumStation    := slotIndex + 1;    // configured for GetSignalStr
	GetSignalStr_0.uNumSignal     := j + 1;		    // configured for GetSignalStr

	GetSignalStr_0();
	GetSignalStr_1();

END_PROGRAM

PROGRAM _CYCLIC
	//-----------------------------------------------------------------
	// This program can be used for I/O forcing
	// The variable slotIndex should mapped to I/O module selection
	// in the HMI. That is, slotIndex = 0 is your first module in
	// the HW configuration. Furthermore you should map ForceValue
	// and ForceStatus variables to corresponding module layers
	// respectively. As an example, your HMI should look like as
	// Module's I/O mapping page in monitor mode; that is, a selection
	// box to represent ForceStatus and then a ForceValue input...
	//
	// The FB BuildSignalStr; builds the specific channel address
	// string according to the selection made from the HMI
    //
	// MAX_DP_INDEX should be configured. It is the number of channels
	// on the selected IO card (e.g. There are 12 channels on X20 DO9322
	// thus the value for MAX_DP_INDEX should be 11)
	//
	// The program will automatically do everything according to the
	// selection made from the HMI.
	//
	//-----------------------------------------------------------------
	// abdullahoglf, 20.12.2013
	//-----------------------------------------------------------------

	//-----------------------------------
	// Get cmd from the HMI
	HMImap;

	// DI card
	IF (slotIndex + ioCfgStart) >= diStartIndex AND (slotIndex + ioCfgStart <= diStartIndex + diCount - 1) THEN
		GetSignalStr_0.eTypeSignal  := DI_IO;
		GetSignalStr_1.eTypeSignal  := DI_IO;
		MAX_DP_INDEX := 15;

		// DO card
	ELSIF (slotIndex + ioCfgStart) >= doStartIndex AND (slotIndex + ioCfgStart <= doStartIndex + doCount - 1) THEN
		GetSignalStr_0.eTypeSignal  := DO_IO;
		GetSignalStr_1.eTypeSignal  := DO_IO;
		MAX_DP_INDEX := 15;

		// AO card
	ELSIF (slotIndex + ioCfgStart) >= aoStartIndex AND (slotIndex + ioCfgStart <= aoStartIndex + aoCount - 1) THEN
		GetSignalStr_0.eTypeSignal  := AO_IO;
		GetSignalStr_1.eTypeSignal  := AO_IO;
		MAX_DP_INDEX := 1;

		// AI card
	ELSIF (slotIndex + ioCfgStart) >= aiStartIndex AND (slotIndex + ioCfgStart <= aiStartIndex + aiCount - 1) THEN
		GetSignalStr_0.eTypeSignal  := AI_IO;
		GetSignalStr_1.eTypeSignal  := AI_IO;
		// AI2632 has two input channels
		IF slotIndex + ioCfgStart = aoStartIndex - 1 THEN
			MAX_DP_INDEX := 1;
		ELSE
			MAX_DP_INDEX := 1;
		END_IF;

	END_IF;

	GetSignalStr_0();
	GetSignalStr_1();
	(* ------------------------------------------------------------------ *)
	(*  ----------------------     MAIN CONTROL     --------------------- *)
	(*  ----------------------------------------------------------------- *)
	HMIforceStep:= forceStep;
	CASE forceStep OF
		FORCE_WAIT:
			IF NOT loopBypass THEN
				// Check if the force should be activated
				FOR i := 0 TO 15 DO
					// Give the command for forcing if the request is done from the Visu
					IF ForceHandle.Status.ModuleForceStatus[slotIndex].ForceStatus[i] = 1 AND ForceHandle.Status.ModuleForceStatus[slotIndex].ForceStatusOld[i] = 0 THEN
						ForceHandle.Status.ModuleForceStatus[slotIndex].ForceStatusOld[i] := ForceHandle.Status.ModuleForceStatus[slotIndex].ForceStatus[i];
						ForceHandle.Cmd.Force                                             := TRUE;
						loopBypass                                                        := TRUE;
						EXIT;
					END_IF;

				END_FOR;
			END_IF;

			IF NOT loopBypass THEN
				// Check if the force should be deactivated
				FOR i := 0 TO 15 DO
					// Give the command for forcing if the request is done from the Visu
					IF ForceHandle.Status.ModuleForceStatus[slotIndex].ForceStatus[i] = 0 AND ForceHandle.Status.ModuleForceStatus[slotIndex].ForceStatusOld[i] = 1 THEN
						ForceHandle.Status.ModuleForceStatus[slotIndex].ForceStatusOld[i] := ForceHandle.Status.ModuleForceStatus[slotIndex].ForceStatus[i];
						ForceHandle.Cmd.DisableForce                                      := TRUE;
						loopBypass                                                        := TRUE;
						EXIT;
					END_IF;

				END_FOR;
			END_IF;

			IF NOT loopBypass THEN
				// Check the force values from the HMI; if there is a change and the realted channel is forced, write it to the channel
				FOR i := 0 TO 15 DO
					IF ((ForceHandle.Status.ModuleForceStatus[slotIndex].ForceValue[i] <> ForceHandle.Status.ModuleForceStatus[slotIndex].ForceValueOld[i]) AND
						ForceHandle.Status.ModuleForceStatus[slotIndex].IsForced[i] = TRUE) THEN
						ForceHandle.Status.ModuleForceStatus[slotIndex].ForceValueOld[i] := ForceHandle.Status.ModuleForceStatus[slotIndex].ForceValue[i];
						ForceHandle.Cmd.WriteForceValue := TRUE;
						loopBypass                      := TRUE;

						//-------- configure GetSignalStr ------
						GetSignalStr_0.uNumStation  := slotIndex + 1;    // configured for GetSignalStr
						GetSignalStr_0.uNumSignal   := i + 1;		     // configured for GetSignalStr

						GetSignalStr_0();
						//---------------------------------------

						EXIT;
					END_IF;

				END_FOR;
			END_IF;

			// Enable forcing for a specific channel
			IF ForceHandle.Cmd.Force THEN
				ForceHandle.Cmd.Force := FALSE;

				//-------- configure GetSignalStr ------
				GetSignalStr_0.uNumStation  := slotIndex + 1;    // configured for GetSignalStr
				GetSignalStr_0.uNumSignal   := i + 1;		     // configured for GetSignalStr

				GetSignalStr_0();
				//---------------------------------------

				// datapoint of the channel is already known
				EnableIOForcing.pDatapoint := ADR(GetSignalStr_0.sStrSignal);
				EnableIOForcing.enable     := TRUE;
				forceStep               := FORCE_ENABLE_FORCE;

				// write the force value
			ELSIF ForceHandle.Cmd.WriteForceValue THEN
				ForceHandle.Cmd.WriteForceValue := FALSE;
				SetForceValue.enable            := TRUE;
				SetForceValue.pDatapoint        := ADR(GetSignalStr_0.sStrSignal);
				SetForceValue.value             := ForceHandle.Status.ModuleForceStatus[slotIndex].ForceValue[i];
				forceStep                    := FORCE_WRITE;

				// Disable forcing for a specific channel
			ELSIF ForceHandle.Cmd.DisableForce THEN
				ForceHandle.Cmd.DisableForce := FALSE;
				//-------- configure GetSignalStr ------
				GetSignalStr_0.uNumStation  := slotIndex + 1;    // configured for GetSignalStr
				GetSignalStr_0.uNumSignal   := i + 1;		      // configured for GetSignalStr

				GetSignalStr_0();
				//---------------------------------------
				forceStep               := FORCE_DISABLE_SPECIFIC_FORCE;

				// Disable global forcing
			ELSIF ForceHandle.Cmd.DisableForceGlobal THEN
				ForceHandle.Cmd.DisableForceGlobal := FALSE;
				DisableAllForcing.enable           := TRUE;
				forceStep                       := FORCE_DISABLE_ALL;
			END_IF;

			//----------------------------------------------
			// Enable Forcing for a specific datapoint
		FORCE_ENABLE_FORCE:
			IF EnableIOForcing.status = ERR_OK AND NOT ForceHandle.Cmd.WriteForceValue THEN	// FB completed w/o an error
				EnableIOForcing.enable                                       := FALSE;
				ForceHandle.Status.ModuleForceStatus[slotIndex].IsForced[i]  := TRUE;
				forceStep              								         := FORCE_WAIT;

			ELSIF EnableIOForcing.status = ERR_OK AND ForceHandle.Cmd.WriteForceValue THEN  // FB completed w/o an error, forcing is in progress
				EnableIOForcing.enable                                            := FALSE;
				ForceHandle.Status.ModuleForceStatus[slotIndex].IsForced[i]       := TRUE;
				ForceHandle.Status.ModuleForceStatus[slotIndex].ForceStatus[i]    := TRUE;
				ForceHandle.Status.ModuleForceStatus[slotIndex].ForceStatusOld[i] := ForceHandle.Status.ModuleForceStatus[slotIndex].ForceStatus[i];
				SetForceValue.enable                                              := TRUE;
				SetForceValue.pDatapoint                                          := lastDataPoint;
				SetForceValue.value                                               := ForceHandle.Status.ModuleForceStatus[slotIndex].ForceValue[i];
				ForceHandle.Cmd.WriteForceValue                                   := FALSE;
				forceStep                                                         := FORCE_WRITE;

			ELSIF EnableIOForcing.status <> ERR_OK AND EnableIOForcing.status <> ERR_FUB_BUSY THEN // FB completed w/ an error
				forceErrorID           := EnableIOForcing.status;
				forceWaitMsg           := 'FORCE_ENABLE_FORCE - Something went wrong during trying to force';
				EnableIOForcing.enable := FALSE;
				TEST_INT			:= 10;
				forceStep           := FORCE_ERROR;
			END_IF;

			//----------------------------------------------
			// Write the forcing value
		FORCE_WRITE:
			IF SetForceValue.status = ERR_OK THEN   // FB completed w/o an error
				SetForceValue.enable := FALSE;
				forceStep            := FORCE_WAIT;

			ELSIF SetForceValue.status <> ERR_OK AND SetForceValue.status <> ERR_FUB_BUSY THEN  // FB completed w/ an error
				SetForceValue.enable := FALSE;
				forceWaitMsg         := 'FORCE_WRITE - Something went wrong while writing the force value';
				forceErrorID         := SetForceValue.status;
				TEST_INT			:= 20;
				forceStep            := FORCE_ERROR;
			END_IF;

			//----------------------------------------------
			// Disable Forcing for a specific datapoint
		FORCE_DISABLE_SPECIFIC_FORCE:
			DisableForcing.enable      := TRUE;
			DisableForcing.pDatapoint  := ADR(GetSignalStr_0.sStrSignal);
			IF DisableForcing.status = ERR_OK THEN	// FB completed w/o an error
				DisableForcing.enable := FALSE;
				forceStep             := FORCE_WAIT;
				ForceHandle.Status.ModuleForceStatus[slotIndex].IsForced[i]       := FALSE;  // reset the module forced flag
				ForceHandle.Status.ModuleForceStatus[slotIndex].ForceStatus[i]    := 0;

			ELSIF DisableForcing.status <> ERR_OK AND DisableForcing.status <> ERR_FUB_BUSY AND DisableForcing.status <> ERR_FUB_ENABLE_FALSE THEN // FB completed w/ an error
				forceWaitMsg := 'FORCE_DISABLE_SPECIFIC_FORCE - Something went wrong disabling specific forcing';
				forceErrorID := DisableForcing.status;
				TEST_INT			:=30;
				forceStep    := FORCE_ERROR;
			END_IF;

			//----------------------------------------------
			// Disable Forcing globally
		FORCE_DISABLE_ALL:
			IF DisableAllForcing.status = ERR_OK THEN     // FB completed w/o an error
				DisableAllForcing.enable := FALSE;
				FOR slotIndex := 0 TO NUMBER_OF_MODULES_MINUS_ONE DO
					FOR i := 0 TO 15 DO
						ForceHandle.Status.ModuleForceStatus[slotIndex].IsForced[i]       := FALSE;
						ForceHandle.Status.ModuleForceStatus[slotIndex].ForceStatus[i]    := 0;
						ForceHandle.Status.ModuleForceStatus[slotIndex].ForceStatusOld[i] := 0;
					END_FOR;
				END_FOR;

				slotIndex    := 0;
				forceStep    := FORCE_WAIT;

			ELSIF DisableAllForcing.status <> ERR_OK AND DisableAllForcing.status <> ERR_FUB_BUSY THEN // FB completed w/ an error
				forceWaitMsg := 'FORCE_DISABLE_ALL - Something went wrong during disabling forcing globally';
				forceErrorID := DisableAllForcing.status;

				TEST_INT			:=40;
				forceStep    := FORCE_ERROR;
			END_IF;

			//----------------------------------------------
			// Error state
		FORCE_ERROR:
			// Disable all the user commands & FB enables
			ForceHandle.Cmd.DisableForce       := FALSE;
			ForceHandle.Cmd.DisableForceGlobal := FALSE;
			ForceHandle.Cmd.Force              := FALSE;

			EnableIOForcing.enable             := FALSE;
			GetIOListDP.enable                 := FALSE;
			DisableAllForcing.enable           := FALSE;
			DisableForcing.enable              := FALSE;

			// Reset the error ID and error msg upon acknowledgement and go back to FORCE_WAIT
			IF ForceHandle.Cmd.ErrAck THEN
				// reset the cmd's
				ForceHandle.Cmd.ErrAck             := FALSE;
				ForceHandle.Cmd.DisableForce       := FALSE;
				ForceHandle.Cmd.DisableForceGlobal := FALSE;
				ForceHandle.Cmd.Force              := FALSE;
				ForceHandle.Cmd.WriteForceValue    := FALSE;
				// Reset variables for GetSignalStr
				GetSignalStr_0.uNumSignal := 0;
				GetSignalStr_0();
				// Reset error msg & program step
				forceWaitMsg           := ' ';
				forceErrorID           := 0;
				forceStep              := FORCE_WAIT;

				// Reset force statuses
				FOR slotIndex := 0 TO NUMBER_OF_MODULES_MINUS_ONE DO
					FOR i := 0 TO 15 DO
						ForceHandle.Status.ModuleForceStatus[slotIndex].IsForced[i]       := FALSE;
						ForceHandle.Status.ModuleForceStatus[slotIndex].ForceStatus[i]    := FALSE;
						ForceHandle.Status.ModuleForceStatus[slotIndex].ForceStatusOld[i] := ForceHandle.Status.ModuleForceStatus[slotIndex].ForceStatus[i];
					END_FOR;
				END_FOR;
				// Reset the HMI selection variable
				slotIndex := 0;
				i         := 0;
			END_IF;
	END_CASE;

	IF forceStep <> FORCE_WAIT AND loopBypass THEN
		loopBypass := FALSE;
	END_IF;

	//Check if error is active - flag is used in HMI for color datapoint of status text
	IF(forceStep = FORCE_ERROR)THEN
		ForceHandle.Status.ErrorActive := 1;
	ELSE
		ForceHandle.Status.ErrorActive := 0;
	END_IF

	(******************	             FB CALLS                  *****************)
	GetIOListDP();
	EnableIOForcing();
	DisableForcing();
	DisableAllForcing();
	SetForceValue();

//	IF NOT gSimulation THEN
		GetPhsyicalStatus;  // call the action to see the physical statuses of the datapoints
//	END_IF;

END_PROGRAM
```

#### Types.typ - Local data types
```iecst
(********************************************************************
 * COPYRIGHT -- Bernecker + Rainer
 ********************************************************************
 * Program: ForceIO
 * File: ForceIO.typ
 * Author: abdullahoglf
 * Created: December 18, 2013
 ********************************************************************
 * Local data types of program ForceIO
 ********************************************************************)

TYPE
	Status_typ : 	STRUCT
		ModuleForceStatus : ARRAY[0..NUMBER_OF_MODULES_MINUS_ONE]OF ForceStatus_typ;
		ErrorActive : USINT; (*Flag that error is active*)
	END_STRUCT;
	ForceStatus_typ : 	STRUCT
		ForceValueOld : ARRAY[0..15]OF UDINT; (*Force value from the HMI from the previous cycle*)
		ForceValue : ARRAY[0..15]OF UDINT; (*Force value from the HMI*)
		ForceStatusOld : ARRAY[0..15]OF BOOL; (*Represents the force status request from the HMI of the related I/O channel from previous cycles*)
		ForceStatus : ARRAY[0..15]OF BOOL; (*Represents the current force status request from the HMI of the related I/O channel*)
		IsForced : ARRAY[0..15]OF BOOL; (*Represents the current force status of the channel*)
	END_STRUCT;
	ForceModuleParameter_typ : 	STRUCT
		DatapointToControl : ARRAY[0..15]OF UDINT;
	END_STRUCT;
	ForceParameters_typ : 	STRUCT
		ModuleForceParameter : ARRAY[0..NUMBER_OF_MODULES_MINUS_ONE]OF ForceModuleParameter_typ;
	END_STRUCT;
	ForceCmd_typ : 	STRUCT
		ErrAck : BOOL; (*Error Acknowledge*)
		GetStatus : BOOL; (*Cmd to get the status*)
		DisableForceGlobal : BOOL; (*Disables forcing for all channels*)
		WriteForceValue : BOOL; (*Cmd to write the force value to the channel*)
		DisableForce : BOOL; (*Disables forcing for a specific channel*)
		Force : BOOL; (*Enables forcing for a specific channel*)
	END_STRUCT;
	ForceHandle_typ : 	STRUCT
		Cmd : ForceCmd_typ;
		Status : Status_typ;
		Parameters : ForceParameters_typ;
	END_STRUCT;
	GetStatus_enm :
		(
		STATUS_ERROR,
		STATUS_GET_STATUS,
		STATUS_WAIT
		);
	ForceStep_enm :
		(
		FORCE_WAIT := 0,
		FORCE_ENABLE_FORCE := 10,
		FORCE_WRITE := 20,
		FORCE_DISABLE_SPECIFIC_FORCE := 30,
		FORCE_DISABLE_ALL := 40,
		FORCE_ERROR := 99
		);
END_TYPE
```

#### Variables.var - Local variables
```iecst
(********************************************************************
 * COPYRIGHT -- Bernecker + Rainer
 ********************************************************************
 * Program: ForceIO
 * File: ForceIO.var
 * Author: abdullahoglf
 * Created: December 18, 2013
 ********************************************************************
 * Local variables of program ForceIO
 ********************************************************************)
VAR
	ForceHandle : ForceHandle_typ := (0); (*Force I/O task handle*)
	HMIforceStep : DINT;
	forceStep : ForceStep_enm; (*States for the program*)
	forceWaitMsg : STRING[100]; (*Error msg from the task*)
	i : USINT; (*Iteration variable*)
	k : USINT := 0; (*Iteration variable*)
	t : USINT; (*Iteration variable*)
	j : USINT; (*Iteration variable*)
	lastDataPoint : UDINT; (*Datapoint found by GetIOList*)
	forceErrorID : UINT; (*Development diagnostics based error ID*)
END_VAR
(*==========================         Function Blocks           ==============================*)
VAR
	GetSignalStr_1 : BuildSignalStr := (0);
	GetSignalStr_0 : BuildSignalStr := (0);
	GetDPStatus : AsIODPStatus := (0); (*FB to see the physical value of the I/O datapoint*)
	SetForceValue : AsIOSetForceValue; (*FB to set force value*)
	EnableIOForcing : AsIOEnableForcing; (*FB to enable frocing*)
	GetIOListDP : AsIOListDP; (*FB to get the IO address list*)
	DisableAllForcing : AsIOGlobalDisableForcing := (0); (*FB to disable forcing for all channels*)
	DisableForcing : AsIODisableForcing; (*FB to disable specific channel*)
END_VAR
(*=========================         Variables for GetSignalStr Action    =====================*)
VAR
	slotIndex : USINT; (*Slot number iteration variable*)
	loopBypass : BOOL; (*Flag to bypass to loops*)
END_VAR
(*==========================                    Constants           ==============================									*)
VAR
	TEST_INT : INT;
	MAX_DP_INDEX : USINT := 0; (*Max datapoint index in an IO card -- depends on the type of the card*)
END_VAR
```

#### ForceIO_Actions.st
```iecst
(********************************************************************
 * COPYRIGHT -- Bernecker + Rainer
 ********************************************************************
 * Program: ForceIO
 * File: ForceIO_Actions.st
 * Author: abdullahoglf
 * Created: January 15, 2014
 *******************************************************************)

(* Comm with the HMI *)
ACTION HMImap:

	// Assign max. number of chanels in curent card
	gHMI.IO_Control.MaxDpIndex := MAX_DP_INDEX;

	IF slotIndex = gHMI.IO_Control.SelectedSlotOld THEN
		FOR j := 0 TO 15 DO
			ForceHandle.Status.ModuleForceStatus[slotIndex].ForceStatus[j]    := gHMI.IO_Control.ForceStatus[j];
			ForceHandle.Status.ModuleForceStatus[slotIndex].ForceValue[j]     := gHMI.IO_Control.FoceValue[j];
		END_FOR;
	END_IF;

	//----------------------------
	// Reset the cmd's if the user
	// changes the active slot
	IF slotIndex <> gHMI.IO_Control.SelectedSlotOld THEN
		k  := 0;  // iteration variable for status monitoring is reset
		FOR j := 0 TO 15 DO
			gHMI.IO_Control.FoceValue[j]                                      := ForceHandle.Status.ModuleForceStatus[slotIndex].ForceValueOld[j];
			gHMI.IO_Control.ForceStatus[j]                                    := ForceHandle.Status.ModuleForceStatus[slotIndex].ForceStatusOld[j];
			ForceHandle.Status.ModuleForceStatus[slotIndex].ForceStatus[j]    := gHMI.IO_Control.ForceStatus[j];
			ForceHandle.Status.ModuleForceStatus[slotIndex].ForceValue[j]     := gHMI.IO_Control.FoceValue[j];

			ForceHandle.Status.ModuleForceStatus[slotIndex].ForceStatusOld[j] := ForceHandle.Status.ModuleForceStatus[slotIndex].ForceStatus[j];
			ForceHandle.Status.ModuleForceStatus[slotIndex].ForceValueOld[j]  := ForceHandle.Status.ModuleForceStatus[slotIndex].ForceValue[j];
		END_FOR;

	END_IF;

END_ACTION

(* Gets the physical status of the I/O datapoints *)
ACTION GetPhsyicalStatus:
	IF GetDPStatus.status <> ERR_OK AND GetDPStatus.status <> ERR_FUB_BUSY AND GetDPStatus.status <> ERR_FUB_ENABLE_FALSE THEN
		GetDPStatus.enable := FALSE;
		k                  := 0;     // reset the channel index in case of any error
	ELSE
		GetDPStatus.enable := TRUE;
	END_IF;

	GetDPStatus.pDatapoint := ADR(GetSignalStr_1.sStrSignal);

	// FB completed w/o an error
	IF GetDPStatus.status = ERR_OK THEN

		IF (GetDPStatus.flags AND (2#0000_0100)) = 0 THEN  // the datapoint is not forced
			gHMI.IO_Control.PhysicalStatus[k] := GetDPStatus.value;

		ELSE   // the datapoint is forced, map the forced value
			gHMI.IO_Control.PhysicalStatus[k] := GetDPStatus.forceValue;
		END_IF;

		IF k <> MAX_DP_INDEX THEN
			k := k + 1;

		ELSE
			k := 0;
		END_IF;

		//-------- configure GetSignalStr ------
		GetSignalStr_1.uNumStation  := slotIndex + 1;    // configured for GetSignalStr
		GetSignalStr_1.uNumSignal   := k + 1;		     // configured for GetSignalStr

		GetSignalStr_1();
		//---------------------------------------
	END_IF;

	// reset the physical value if the DP is not existing
	FOR t := 0 TO 15 DO
		IF t > MAX_DP_INDEX THEN
			gHMI.IO_Control.PhysicalStatus[t] := 0;
		END_IF;
	END_FOR;

	GetDPStatus();

END_ACTION
```

### Program Logical/SourceCode/Infastructure/ForceIOs/aIOhand (IEC)

#### Variables.var
```iecst
VAR
	TON_0 : TON := (0); (*Help timer*)
	checkName : REFERENCE TO STRING[1]; (*Pointer to access to the IO Name*)
END_VAR
VAR CONSTANT
	MAX_UDINT_NUMBER : UDINT := 4294967295;
END_VAR
```

#### Main.st
```iecst
(********************************************************************
 * COPYRIGHT -- Bernecker + Rainer
 ********************************************************************
 * Program: aIOhand
 * File: aIOhand.st
 * Author: abdullahoglf
 * Created: February 11, 2014
 ********************************************************************
 * Implementation of program aIOhand
 ********************************************************************)

(*********************************************************************************
*With this software various informations about the modules can be obtained.
 detailed expression can be found on help in the path: Programming/Libraries/
 Direct I/O Access AsIODiag.
*Also a list can automatically be created with the desired values. For instance;
 if in the list the variable moduleState is 1, it means that the specified hardware
 is only configured but not included in the hardware; so on and so forth.
*********************************************************************************)

PROGRAM _INIT

	TON_0.IN := TRUE;
	TON_0.PT :=  T#5s;
END_PROGRAM

PROGRAM _CYCLIC

	(*There are seven cases in the software. These respectively are:
		MAIN: Main state is from where the other cases are managed. Also after an error case, the state is switched back to the MAIN again.
	    CREATE_INFO: This is the case where the function DiagCreateInfo() is used.
					DiagCreateInfo(): Collects information about currently configured and/or inserted hardware modules.
		DISPOSE_INFO: This is the case where the function DiagDisposeInfo() is used.
					DiagDisposeInfo(): Frees up the resources taken up by DiagCreateInfo().
		GET_NUM_INFO: This is the case where the function DiagGetNumInfo() is used.
					DiagGetNumInfo(): Reads the numeric value of a specified information entry.
		GET_STR_INFO: This is the case where the function DiagGetStrInfo() is used.
					DiagGetStrInfo(): Reads the string value of a specified information entry.
	    GET_LIST: This case handles the list creating.
	    ERROR: At this case, an error flag is put and upon error acknowledgemnt it then switches the state back to MAIN.
     *)

	CASE state OF

		//-------------------------
		//Wait before starting
		WAIT_START:
			// Wait few seconds after PLC boots up also for a motion to be in RUN

			IF(TON_0.Q)THEN // HMI is out of Init paga and minimum (5s time is elapsed)
				TON_0.IN  := FALSE; 	// reset timer
				state	  := MAIN;		// Change state
				GetList.GetList := TRUE;//NOT(gSimulation);	// Give commad to get list of HW modules
			END_IF

			//-------------------------
			// Ready for cmd's
		MAIN:
			IF  (CreateInfoCommand.createInfo <> FALSE) THEN       //According to the command, the state is decided
				state := CREATE_INFO;
			ELSIF (DisposeInfoCommand.disponseInfo <> FALSE) THEN
				state := DISPOSE_INFO;
			ELSIF (GetNumInfoCommand.getNumInfo <> FALSE) THEN
				state := GET_NUM_INFO;
			ELSIF (GetStrInfoCommand.getStrInfo <> FALSE) THEN
				state := GET_STR_INFO;
				//Process for auto-list generation is initiliazed
			ELSIF (GetList.GetList <> FALSE) THEN
				MyDiagCreateInfo.infoKind := asdiagALL;  //asdiagALL for information about inserted and configured modules
				state                     := CREATE_INFO;
			END_IF;

			//-------------------------
			// Create the information which later on is to be used by other FB's
		CREATE_INFO:
			MyDiagCreateInfo.enable := TRUE;
			MyDiagCreateInfo();
			//If run manually then the function waits for the configuration to be made
			IF (CreateInfoCommand.plugged) THEN
				MyDiagCreateInfo.infoKind := asdiagPLUGGED;
			ELSIF (CreateInfoCommand.configured) THEN
				MyDiagCreateInfo.infoKind := asdiagCONFIGURED;
			ELSIF (CreateInfoCommand.all) THEN
				MyDiagCreateInfo.infoKind := asdiagALL;
			END_IF;

			//If the FB is finished then resettings are done
			IF (MyDiagCreateInfo.status = ERR_OK) THEN
				Info.Ident	   			            := MyDiagCreateInfo.ident;
				Info.NumbersEntries    			    := MyDiagCreateInfo.nrEntries;
				MyDiagCreateInfo.enable             := FALSE;
				CreateInfoCommand.createInfo        := FALSE;
				//If an auto-list generation is progress, the state is transferred to GET_NUM_INFO
				IF (GetList.GetList = TRUE) THEN
					state := GET_NUM_INFO;
					//If otherwise, it goes back to the MAIN and waits
				ELSE
					state := MAIN;
				END_IF;

			ELSIF MyDiagCreateInfo.status = ERR_FUB_BUSY THEN		//Not complete, call it again
				state := CREATE_INFO;
			ELSE
				state := ERROR;
			END_IF

			//---------------------------
			// Release the used handles
		DISPOSE_INFO:
			MyDiagDisposeInfo.enable := TRUE;
			MyDiagDisposeInfo.ident  := Info.Ident;
			MyDiagDisposeInfo();
			//If the FB is completed then it goes back to the MAIN state
			IF MyDiagDisposeInfo.status = ERR_OK THEN
				MyDiagDisposeInfo.enable         := FALSE;
				DisposeInfoCommand.disponseInfo  := FALSE;
				state 							 := MAIN;
				//If not it is called again
			ELSIF MyDiagDisposeInfo.status = ERR_FUB_BUSY THEN
				state := DISPOSE_INFO;
			ELSE
				state := ERROR;
			END_IF;

			//--------------------------
			// Get numeric info. about the IO's
		GET_NUM_INFO:
			MyDiagGetNumInfo.enable   := TRUE;
			MyDiagGetNumInfo.ident    := Info.Ident;
			MyDiagGetNumInfo.infoCode := asdiagMODUL_STATE;
			MyDiagGetNumInfo.index    := Info.Index;
			MyDiagGetNumInfo();
			//If the function is completeand the output setting the resettings are done
			IF MyDiagGetNumInfo.status = 0 THEN
				GetNumInfoCommand.desiredNum := MyDiagGetNumInfo.value;
				MyDiagGetNumInfo.enable      := FALSE;
				GetNumInfoCommand.getNumInfo := FALSE;
				//If a auto-list generation is in progress it continues to GET_STR_INFO
				IF GetList.GetList THEN
					state := GET_STR_INFO;
					//If not, the state is switched back to MAIN
				ELSE
					state := MAIN;
				END_IF;
				//If it is not completed then it is called again
			ELSIF MyDiagGetNumInfo.status = ERR_FUB_BUSY THEN
				state := GET_NUM_INFO;
			ELSE
				state := ERROR;
			END_IF;

			//-----------------------------
			// Get str. info. about the IO's
		GET_STR_INFO:
			MyDiagGetStrInfo.enable    := TRUE;
			MyDiagGetStrInfo.ident     := Info.Ident;
			MyDiagGetStrInfo.index     := Info.Index;
			MyDiagGetStrInfo.infoCode  := asdiagPLUGGED_MODULE;      // for hardware module name
			MyDiagGetStrInfo.pBuffer   := ADR(GetStrInfoCommand.desiredStr);
			MyDiagGetStrInfo.bufferLen := SIZEOF(GetStrInfoCommand.desiredStr);
			MyDiagGetStrInfo();
			IF MyDiagGetStrInfo.status = ERR_OK AND GetList.GetList THEN
				GetStrInfoCommand.getStrInfo         := FALSE;
				MyDiagGetStrInfo.enable              := FALSE;

				//If GetList is enabled then it writes the related values to the list index
				// Check the boundries of GetList array size to avodi writing outside of array
				IF(Info.Index <= (SIZEOF(GetList.List)/ ( SIZEOF(GetList.List[0]) - 1 )) ) THEN // GetList.List size is big enough
					GetList.List[Info.Index].index       := Info.Index;
					GetList.List[Info.Index].name        := GetStrInfoCommand.desiredStr;
					GetList.List[Info.Index].moduleState := GetNumInfoCommand.desiredNum;
					state                                := GET_LIST;
					// Reset IO card positions when entering the GET_LIST step for the first time
					// LT 20140702
					IF(Info.Index = 0)THEN
						diCount 	 := 0;	doCount		 := 0;
						aoCount		 := 0;	aiCount		 := 0;
						diStartIndex := 0;	doStartIndex := 0;
						aiStartIndex := 0;	aoStartIndex := 0;
						ioCfgStart	 := 0;
					END_IF
				ELSE	// Error - GetList.List is smaller than current Info.Index
					state				:= ERROR;	// Go to error state
					brsstrcpy(ADR(Info.errorStatement),ADR('Error - GET_STR_INFO - GetList.List Array too small')); // Give error msg
				END_IF

			ELSIF MyDiagGetStrInfo.status = ERR_OK THEN
				//If not then goes back to the MAIN state
				GetStrInfoCommand.getStrInfo         := FALSE;
				MyDiagGetStrInfo.enable              := FALSE;
				state                                := MAIN;
			ELSIF MyDiagGetStrInfo.status = ERR_FUB_BUSY THEN  //If not completed then it is called again
				state := GET_STR_INFO;
			ELSE
				state := ERROR;
			END_IF;

			//----------------------------
			// Create the list
		GET_LIST:
			// access to IO type definition
			checkName ACCESS (ADR(GetList.List[Info.Index].name) + 3);

			// DI card
			IF brsmemcmp(ADR(checkName), ADR('DI'), SIZEOF(checkName)) = 0 THEN
				IF diCount = 0 THEN
					diStartIndex := Info.Index;
				END_IF;

				diCount := diCount + 1;

				// DO card
			ELSIF brsmemcmp(ADR(checkName), ADR('DO'), SIZEOF(checkName)) = 0 THEN
				IF doCount = 0 THEN
					doStartIndex := Info.Index;
				END_IF;

				doCount := doCount + 1;

				// AI card
			ELSIF brsmemcmp(ADR(checkName), ADR('AI'), SIZEOF(checkName)) = 0 THEN
				IF aiCount = 0 THEN
					aiStartIndex := Info.Index;
				END_IF;

				aiCount := aiCount + 1;

				// AO card
			ELSIF brsmemcmp(ADR(checkName), ADR('AO'), SIZEOF(checkName)) = 0 THEN
				IF aoCount = 0 THEN
					aoStartIndex := Info.Index;
				END_IF;

				aoCount := aoCount + 1;
			END_IF;

			//Index is incremented to fill the list.
			Info.Index := Info.Index+1;

			//When the final value is reached; GetList and index are reset and then DiagDisposeInfo() is run to release the data that has been used.
			IF Info.Index = Info.NumbersEntries THEN
				Info.Index      := 0;
				GetList.GetList := FALSE;
				ioCfgStart      := MIN(MIN(diStartIndex + MAX_UDINT_NUMBER, doStartIndex + MAX_UDINT_NUMBER), MIN(aiStartIndex + MAX_UDINT_NUMBER, aoStartIndex + MAX_UDINT_NUMBER)) + 1;
				state           := DISPOSE_INFO;
			END_IF;

			state := MAIN;

			//----------------------------
			// Error
		ERROR:
			Info.errorFlag := TRUE;
			IF ( 0 = brsstrcmp(ADR(Info.errorStatement), ADR('')) )  THEN
				Info.errorStatement := 'Error! Check statuses of function blocks.';
			END_IF;

			IF Info.errorAck THEN
				// reset the error flag
				Info.errorAck       := FALSE;
				Info.errorFlag      := FALSE;
				Info.errorStatement := '';
				//
				// reset the user cmd's
				GetStrInfoCommand.getStrInfo    := FALSE;
				GetNumInfoCommand.getNumInfo    := FALSE;
				CreateInfoCommand.createInfo    := FALSE;
				DisposeInfoCommand.disponseInfo := FALSE;
				GetList.GetList                 := FALSE;
				//
				// reset the FB enables
				MyDiagCreateInfo.enable  := FALSE;
				MyDiagGetStrInfo.enable  := FALSE;
				MyDiagGetNumInfo.enable  := FALSE;
				MyDiagDisposeInfo.enable := FALSE;
				//
				// reset the SW step
				state := MAIN;
			END_IF;
	END_CASE;

	// Execute help  timer
	TON_0();

END_PROGRAM
```

### Program Logical/SourceCode/Infastructure/HMI (IEC)

#### Main.st - Init, cyclic, exit code
```iecst
(*********************************************************************************
 * Copyright:
 * Author:    baranc
 * Created:   September 19, 2025/1:33 PM
 *********************************************************************************)

PROGRAM _INIT

	//Loc.OldMaterialNumber	:=	4; //Program ilk açildiginda Ekrana mecvut seçili ilaçin Degerlerini getirmek için.

END_PROGRAM

PROGRAM _CYCLIC
//	//==================================================
//	//	 Ekrana gönderilecek PML,Pos vb degiskenlerin atanmasi
//	//==================================================
//	Status;
//
//
//	//==================================================
//	//		Ekranda kullanilacak Timerlari çagirma ve atama
//	//==================================================
	GenTimer;

//	//==================================================
//	//		Ekranda bulunan widgetlari gizleme
//	//==================================================
	WidgetVisible;

	//==================================================
	//		IO Force kisminin kontrolleri
	//==================================================
	IOcontrolPage;
//
//	//==================================================
//	//		Manuel Eksen Atamalari
//	//==================================================
//	ManuelAxis;
//
	//==================================================
	//		Makine kilitleme sayfasi kontrolleri
	//==================================================
	MachineLockPage;

//	//==================================================
//	//		Manuel Device
//	//==================================================
//
//		ManualDevice;
//
//
//
//
//	//==================================================
//	//		Maximum ve Minimum deđerlerin atanmasý
//	//==================================================
//	MaxMinValue;
//
//
//	//==================================================
//	//		Home Ýţlemleri
//	//==================================================
//
//		Home;
//
//	Hyd;
//
//	SpacerType;
//
//	Distance;
//
//

END_PROGRAM

PROGRAM _EXIT
	(* Insert code here *)

END_PROGRAM
```

#### Types.typ - Local data types
```iecst
TYPE
	LocType : 	STRUCT
		SelectedStatus : LocSelectedStatus;
		FB : LocFBType;
		PowerStatus : BOOL;
		oldEdgeCaptureStep : Step_EC;
		EdgeCaptureStep : Step_EC;
		FirstInStepEC : BOOL;
		oldActiveUnit : INT;
		OldSpacerType : INT;
		OldMaterialNumber : INT;
		ReferenceStatus : BOOL;
	END_STRUCT;
	LocFBType : 	STRUCT
		Timer : LocFBTimerType;
	END_STRUCT;
	LocFBTimerPulseType : 	STRUCT
		ms50 : TON;
		ms100 : TON;
		ms200 : TON;
		ms300 : TON;
		ms500 : TON;
		ms1000 : TON;
	END_STRUCT;
	LocFBTimerType : 	STRUCT
		Pulse : LocFBTimerPulseType;
		TP_MachineReset : TP;
		TON_SubStepTOut : TON;
		TON_State : TON;
		ProcessTime : TIME;
		TON_ProcessTrace : TON;
		TON_VacuumTimeout : TON; (*//bc25.07.07*)
		TON_VacuumWait : TON;
		TON_ProcessTrackingTime : TON;
		TON_Y_ReturnAfterTakingGlass : TON;
		TON_Y_DelaySecond : TON;
		TON_WaitingTimeBeforeMiter : TON;
	END_STRUCT;
	Step_EC :
		(
		EC_WAIT_CMD,
		EC_START,
		EC_OFSET,
		EC_FINISH
		);
	LocSelectedStatus : 	STRUCT
		ExitThicness : BOOL;
		EntryThicness : BOOL;
		Bridges : BOOL;
		Entrys : BOOL;
		ConvWithVacuum : BOOL;
		VacuumWithConv : BOOL;
		Exits : BOOL;
	END_STRUCT;
END_TYPE
```

#### Variables.var - Local variables
```iecst
VAR
	bHMIBigGlass : BOOL;
	bHMIPower : BOOL;
	i : UINT;
	_i : UINT;
	Loc : LocType;
	_k : UINT;
	_j : UINT;
END_VAR
(*Machine Lock Get Time*)
VAR
	SystemTime : DATE_AND_TIME;
	DTGetTime_0 : DTGetTime;
	DTStructureGetTime_0 : DTStructureGetTime;
	DTStructure_0 : DTStructure;
	tempDay : STRING[80];
	tempMonth : STRING[80];
	NormalPassword : STRING[80];
	oldMonth : USINT;
	oldDay : USINT;
	SuperPassword : STRING[80];
	TON_Logout : TON;
	CmsGetTimeStatus : UDINT;
END_VAR
(*test için eklendi *)
VAR
	bTest01 : BOOL;
END_VAR
(*Manual Device FB*)
VAR
	(*fbManualDeviceCtrl : ARRAY[0..Max_Manual_Device] OF fbManualDevice;*)
	MC_ReadParameterZ_FB : MC_ReadParameter;
	MC_ReadParameterC_FB : MC_ReadParameter;
	StateAbsCHomeOffset : INT;
	StateAbsZHomeOffset : INT;
	hmiOldCSetVal : LREAL;
	hmiCSetValSon : LREAL;
	hmiCSetVal : LREAL;
	hmiZSetVal : LREAL;
END_VAR
(*Timers*)
VAR
	TON_ResetAxis : TON;
END_VAR
VAR CONSTANT
	DOWN : USINT := 0;
	UP : USINT := 1;
END_VAR
```

#### ManualDeviceNames.var
```iecst
VAR CONSTANT
	UNIT_LargeSpatulaPiston : USINT := 0;
	UNIT_SmallSpatulaPiston : USINT := 1;
	UNIT_DepthValve : USINT := 2;
	UNIT_MaterialOutValve : USINT := 3;
END_VAR
```

#### WidgetVisible.st
```iecst
ACTION WidgetVisible:

	//======================================
	//			Header Alert Image/Line
	//======================================
	IF gAlert.Abort.Status THEN
		(* Line *)
		gHMI.Widget.AlertLine.Visible := TRUE;

		IF gHMI.Pulse.ms300 THEN
			gHMI.Widget.AlertLine.Style   := 'back_red';
		ELSE
			gHMI.Widget.AlertLine.Style   := 'back_none';
		END_IF;
		(* Image *)

		IF gHMI.CommUnit.ActAlarms > 1 THEN
			gHMI.Widget.AlertImage.Visible := gHMI.Pulse.ms300;
		ELSIF gHMI.CommUnit.ActAlarms <> 0 THEN
			gHMI.Widget.AlertImage.Visible := TRUE;
		END_IF;
		IF gHMI.CommUnit.ActAlarms = 1 THEN
			gHMI.Widget.AlertImage.Image   := 'Media/AlarmX/1.png';
		ELSIF gHMI.CommUnit.ActAlarms = 2 THEN
			gHMI.Widget.AlertImage.Image   := 'Media/AlarmX/2.png';
		ELSIF gHMI.CommUnit.ActAlarms = 3 THEN
			gHMI.Widget.AlertImage.Image   := 'Media/AlarmX/3.png';
		ELSIF gHMI.CommUnit.ActAlarms = 4 THEN
			gHMI.Widget.AlertImage.Image   := 'Media/AlarmX/4.png';
		ELSIF gHMI.CommUnit.ActAlarms = 5 THEN
			gHMI.Widget.AlertImage.Image   := 'Media/AlarmX/5.png';
		ELSIF gHMI.CommUnit.ActAlarms = 6 THEN
			gHMI.Widget.AlertImage.Image   := 'Media/AlarmX/6.png';
		ELSIF gHMI.CommUnit.ActAlarms = 7 THEN
			gHMI.Widget.AlertImage.Image   := 'Media/AlarmX/7.png';
		ELSIF gHMI.CommUnit.ActAlarms = 8 THEN
			gHMI.Widget.AlertImage.Image   := 'Media/AlarmX/8.png';
		ELSE
			gHMI.Widget.AlertImage.Image   := 'Media/AlarmX/9.png';
		END_IF;

	ELSIF gAlert.Stop.Status THEN
		(* Line *)
		gHMI.Widget.AlertLine.Visible := TRUE;

		IF gHMI.Pulse.ms300 THEN
			gHMI.Widget.AlertLine.Style   := 'back_red';
		ELSE
			gHMI.Widget.AlertLine.Style   := 'back_none';
		END_IF;

		(* Image *)
		(*	gHMI.Widget.AlertImage.Visible := gHMI.Pulse.ms300;	*)
		gHMI.Widget.AlertImage.Visible:= TRUE ;
		IF gHMI.CommUnit.ActAlarms = 1 THEN
			gHMI.Widget.AlertImage.Image   := 'Media/AlarmX/1.png';
		ELSIF gHMI.CommUnit.ActAlarms = 2 THEN
			gHMI.Widget.AlertImage.Image   := 'Media/AlarmX/2.png';
		ELSIF gHMI.CommUnit.ActAlarms = 3 THEN
			gHMI.Widget.AlertImage.Image   := 'Media/AlarmX/3.png';
		ELSIF gHMI.CommUnit.ActAlarms = 4 THEN
			gHMI.Widget.AlertImage.Image   := 'Media/AlarmX/4.png';
		ELSIF gHMI.CommUnit.ActAlarms = 5 THEN
			gHMI.Widget.AlertImage.Image   := 'Media/AlarmX/5.png';
		ELSIF gHMI.CommUnit.ActAlarms = 6 THEN
			gHMI.Widget.AlertImage.Image   := 'Media/AlarmX/6.png';
		ELSIF gHMI.CommUnit.ActAlarms = 7 THEN
			gHMI.Widget.AlertImage.Image   := 'Media/AlarmX/7.png';
		ELSIF gHMI.CommUnit.ActAlarms = 8 THEN
			gHMI.Widget.AlertImage.Image   := 'Media/AlarmX/8.png';
		ELSE
			gHMI.Widget.AlertImage.Image   := 'Media/AlarmX/9.png';
		END_IF;

	ELSIF gAlert.Pause.Status THEN
		(* Line *)
		gHMI.Widget.AlertLine.Visible := TRUE;

		IF gHMI.Widget.AlertImage.Visible THEN
			gHMI.Widget.AlertLine.Style   := 'back_orange';
		ELSE
			gHMI.Widget.AlertLine.Style   := 'back_none';
		END_IF;
		(* Image *)
		gHMI.Widget.AlertImage.Visible := gHMI.Pulse.ms300;
		gHMI.Widget.AlertImage.Image   := 'Media/AlarmX/Categories/Category2_Pause.svg';

	ELSIF gAlert.Info.Status THEN
		(* Line *)
		gHMI.Widget.AlertLine.Visible := TRUE;
		IF gHMI.Widget.AlertImage.Visible THEN
			gHMI.Widget.AlertLine.Style   := 'back_blue';
		ELSE
			gHMI.Widget.AlertLine.Style   := 'back_none';
		END_IF;
		(* Image *)
		gHMI.Widget.AlertImage.Visible := TRUE;
		gHMI.Widget.AlertImage.Image   := 'Media/AlarmX/Categories/Category3_Info.svg';

	ELSE
		gHMI.Widget.AlertImage.Image   := 'Media/AlarmX/Categories/Category3_Info.svg';
		gHMI.Widget.AlertLine.Style   := 'back_blue';
		gHMI.Widget.AlertLine.Visible  := FALSE;
		gHMI.Widget.AlertImage.Visible := FALSE;
	END_IF;
END_ACTION
```

#### GenTimer.st
```iecst
(*********************************************************************************
 * Copyright: B&R Industrial Automation GmbH
 * Author:    kay3a
 * Created:   June 24, 2025/9:29 PM
 *********************************************************************************)
ACTION GenTimer:

	//======================================
	//			  Timer Genarate
	//======================================
	(* 50ms *)
	Loc.FB.Timer.Pulse.ms50.PT := T#50ms;
	Loc.FB.Timer.Pulse.ms50.IN := NOT Loc.FB.Timer.Pulse.ms50.Q;
	Loc.FB.Timer.Pulse.ms50();
	IF Loc.FB.Timer.Pulse.ms50.Q THEN
		gHMI.Pulse.ms50 := NOT gHMI.Pulse.ms50;
	END_IF;

	(* 100ms *)
	Loc.FB.Timer.Pulse.ms100.PT := T#100ms;
	Loc.FB.Timer.Pulse.ms100.IN := NOT Loc.FB.Timer.Pulse.ms100.Q;
	Loc.FB.Timer.Pulse.ms100();
	IF Loc.FB.Timer.Pulse.ms100.Q THEN
		gHMI.Pulse.ms100 := NOT gHMI.Pulse.ms100;
	END_IF;

	(* 200ms *)
	Loc.FB.Timer.Pulse.ms200.PT := T#200ms;
	Loc.FB.Timer.Pulse.ms200.IN := NOT Loc.FB.Timer.Pulse.ms200.Q;
	Loc.FB.Timer.Pulse.ms200();
	IF Loc.FB.Timer.Pulse.ms200.Q THEN
		gHMI.Pulse.ms200 := NOT gHMI.Pulse.ms200;
	END_IF;

	(* 300ms *)
	Loc.FB.Timer.Pulse.ms300.PT := T#300ms;
	Loc.FB.Timer.Pulse.ms300.IN := NOT Loc.FB.Timer.Pulse.ms300.Q;
	Loc.FB.Timer.Pulse.ms300();
	IF Loc.FB.Timer.Pulse.ms300.Q THEN
		gHMI.Pulse.ms300 := NOT gHMI.Pulse.ms300;
	END_IF;

	(* 500ms *)
	Loc.FB.Timer.Pulse.ms500.PT := T#500ms;
	Loc.FB.Timer.Pulse.ms500.IN := NOT Loc.FB.Timer.Pulse.ms500.Q;
	Loc.FB.Timer.Pulse.ms500();
	IF Loc.FB.Timer.Pulse.ms500.Q THEN
		gHMI.Pulse.ms500 := NOT gHMI.Pulse.ms500;
	END_IF;

	(* 1000ms *)
	Loc.FB.Timer.Pulse.ms1000.PT := T#1000ms;
	Loc.FB.Timer.Pulse.ms1000.IN := NOT Loc.FB.Timer.Pulse.ms1000.Q;
	Loc.FB.Timer.Pulse.ms1000();
	IF Loc.FB.Timer.Pulse.ms1000.Q THEN
		gHMI.Pulse.ms1000 := NOT gHMI.Pulse.ms1000;
	END_IF;
	//======================================

END_ACTION
```

#### Status.st
```iecst
(*********************************************************************************
 * Copyright: B&R Industrial Automation GmbH
 * Author:    kay3a
 * Created:   June 24, 2025/9:29 PM
 *********************************************************************************)
ACTION Status:

	//======================================
	//		   Cam bekletme istegi.
	//======================================
	IF gFixData.Config.PressTransferPause THEN
		IF gHMI.Pulse.ms300 THEN
			gHMI.Widget.PressGlassPause.Style  := 'Operate';
		ELSE
			gHMI.Widget.PressGlassPause.Style  := 'Operate1';
		END_IF;

	ELSE
		gHMI.Widget.PressGlassPause.Style  := 'Operate1';
	END_IF;

	//======================================
	//		   Reset Butonu istegi gelirse.
	//======================================
	IF (gPML[0].StateCurrent = mpPACKML_STATE_ABORTED OR gPML[0].StateCurrent = mpPACKML_STATE_STOPPED
		OR gAlert.Abort.Status OR gAlert.Stop.Status ) AND gHMI.Pulse.ms100
		THEN
		gHMI.Widget.ResetButton.Style  := 'Operate';
	ELSE
		gHMI.Widget.ResetButton.Style  := 'Operate1';
	END_IF;

	//======================================
	//		   Hareketli eksenleri görelim.
	//======================================
	FOR _k:=0 TO MAX_AX_NR_MIN1 DO
	(*	IF ABS(gAxBasic[_k].Velocity) > 1 THEN*)
	  		gHMI.Diagnosis.Ax[_k].MoveActive := gAxBasic[_k].MoveActive;
//		END_IF;

	END_FOR;
	//======================================
	//		   Tüm PMLleri ekrana gönderelim.
	//======================================
	gIO;
	FOR _k:=0  TO MAX_AX_NR_MIN1 DO
		gHMI.Diagnosis.Ax[_k].Speed := gAxBasic[_k].Velocity;
		gHMI.Diagnosis.Ax[_k].Pos := gAxBasic[_k].Position;
		gHMI.Diagnosis.Ax[_k].HomeStatus := gAxBasic[_k].IsHomed;
		gHMI.Diagnosis.Ax[_k].PowerOn    := gAxBasic[_k].PowerOn;
	END_FOR;
	FOR _k:=0 TO MAX_PML_TASK_NR_MIN1 DO

		gHMI.Status.PML[_k].Name		 := _k;
		gHMI.Status.PML[_k].ModeID 		 := gPML[_k].ModeID;
		gHMI.Status.PML[_k].State 		 := gPML[_k].StateCurrent;
		gHMI.Status.PML[_k].SubState  	 := gPML[_k].SubStateCurrent;
	END_FOR;

	//======================================
	//			REFERANS VE PARK ISLEMLERININ YAPILMA IZNI
	//======================================
	IF gPML[0].StateCurrent <> mpPACKML_STATE_IDLE THEN
		gHMI.Widget.ParkAndRefRequest.Enable := FALSE;
	ELSE
		gHMI.Widget.ParkAndRefRequest.Enable := TRUE;
	END_IF;

	//======================================
	//		   ACT DEPTH VIEW
	//======================================

	gHMI.Diagnosis.Depth.Pos			:= gActDepth;

	//======================================
	//		   Seçili Üniteyi Gösterelim.
	//======================================
	IF gFixData.Config.ActiveUnit = 1 THEN
		gHMI.Widget.Unit1.Style 		 := 'Command';
		gHMI.Widget.Unit2.Style 		 := 'default';
	ELSIF gFixData.Config.ActiveUnit = 2  THEN
		gHMI.Widget.Unit1.Style 		 := 'default';
		gHMI.Widget.Unit2.Style 		 := 'Command';
	END_IF;

	//======================================
	//		  Homing Durumlarýný Görelim
	//======================================
	Loc.ReferenceStatus := TRUE;
	FOR _k :=0 TO MAX_AX_NR_MIN1 DO
		IF gFixData.Ax[_k].Enabled AND gAxBasic[_k].IsHomed THEN
			gHMI.Widget.Ax[_k].Style := 'Command';
		ELSE
			gHMI.Widget.Ax[_k].Style := 'default';
		END_IF;
		IF gFixData.Ax[_k].Enabled AND gAxBasic[_k].IsHomed =FALSE THEN
			Loc.ReferenceStatus:= FALSE;
		END_IF
	END_FOR;

	FOR  _k := EXIT2_UNIT  TO EXIT8_UNIT DO
		gHMI.Diagnosis.Brdige[_k].HomeStatus := fbExitBridgeCtrl_0[_k].Out.Status.Homed;
		IF fbExitBridgeCtrl_0[_k].Out.Status.Homed  AND _k <= gFixData.HwConfig.ExitUnitInstalled THEN
			gHMI.Widget.Bridge[_k].Style := 'Command';

		ELSE
			gHMI.Widget.Bridge[_k].Style := 'default';
		END_IF;
		IF fbExitBridgeCtrl_0[_k].Out.Status.Homed = FALSE  AND _k <= gFixData.HwConfig.ExitUnitInstalled THEN
			Loc.ReferenceStatus:= FALSE;
		END_IF

	END_FOR;
	// giriţ kalýnlýk eksenler home yaptý mý?
	FOR  _k := ENTR1_UNIT  TO ENTR4_UNIT DO
		gHMI.Diagnosis.EntryThickness[_k].HomeStatus := fbEntryZAscMotorCtrl[_k].Out.Status.Homed;
		IF fbEntryZAscMotorCtrl[_k].Out.Status.Homed  AND _k <= gFixData.HwConfig.EntryUnitInstalled THEN
			gHMI.Widget.EntryThickness[_k].Style := 'Command';
		ELSE
			gHMI.Widget.EntryThickness[_k].Style := 'default';
		END_IF;
		IF fbEntryZAscMotorCtrl[_k].Out.Status.Homed = FALSE  AND _k <= gFixData.HwConfig.EntryUnitInstalled THEN
			Loc.ReferenceStatus:= FALSE;
		END_IF

	END_FOR;
	// çýkýţ kalýnlýk eksenler home yaptý mý?
	FOR  _k := EXIT1_UNIT  TO EXIT8_UNIT DO
		gHMI.Diagnosis.ExitThickness[_k].HomeStatus := fbExitZAscMotorCtrl[_k].Out.Status.Homed;
		IF fbExitZAscMotorCtrl[_k].Out.Status.Homed  AND _k <= gFixData.HwConfig.ExitUnitInstalled THEN
			gHMI.Widget.ExitThickness[_k].Style := 'Command';
		ELSE
			gHMI.Widget.ExitThickness[_k].Style := 'default';
		END_IF;
		IF fbExitZAscMotorCtrl[_k].Out.Status.Homed = FALSE  AND _k <= gFixData.HwConfig.ExitUnitInstalled THEN
			Loc.ReferenceStatus:= FALSE;
		END_IF

	END_FOR;

	IF gCommUnit.Main.In.Referance THEN
		IF gHMI.Pulse.ms500 THEN
			gHMI.Widget.PowerGroup.Reference.Style := 'Command';
		ELSE
			gHMI.Widget.PowerGroup.Reference.Style := 'default';
		END_IF

	ELSIF Loc.ReferenceStatus THEN
		gHMI.Widget.PowerGroup.Reference.Style := 'Command';
		gCommUnit.Main.Status.Referenced := TRUE;
	ELSE

		gCommUnit.Main.Status.Referenced := FALSE;
	END_IF;
	//======================================
	//Eksenler Park Pozisyonunda mý ?
	//======================================
	IF gCommUnit.Main.In.Park THEN
		IF gHMI.Pulse.ms300 THEN
			gHMI.Widget.PowerGroup.Park.Style := 'Command';
		ELSE
			gHMI.Widget.PowerGroup.Park.Style := 'default';
		END_IF
	ELSIF gCommUnit.Main.Status.MachineParked THEN
		gHMI.Widget.PowerGroup.Park.Style := 'Command';
	ELSE
		gHMI.Widget.PowerGroup.Park.Style := 'default';
	END_IF;

	//======================================
	//		  Auto Man Durumunu Görelim
	//======================================

	IF gPML[0].ModeID = PML_MODE_MAN THEN
		gHMI.Widget.PowerGroup.Automatic.Style := 'default';
		gHMI.Widget.PowerGroup.Automatic.Enable := TRUE;// manual iken enable olabilsin
		gHMI.Widget.PowerGroup.Manual.Style := 'Command';
	ELSIF gPML[0].ModeID = PML_MODE_AUTO THEN
		gHMI.Widget.PowerGroup.Automatic.Style := 'Command';
		gHMI.Widget.PowerGroup.Manual.Style := 'default';
		gHMI.Widget.PowerGroup.Automatic.Enable := FALSE;
	END_IF;

	//======================================
	//		  Power Durumuu görelim
	//======================================
	Loc.PowerStatus := TRUE;
	FOR _k:=0 TO MAX_AX_NR_MIN1 DO
		IF gFixData.Ax[_k].Enabled  AND gAxBasic[_k].PowerOn =FALSE THEN
			Loc.PowerStatus := FALSE;
			EXIT;
		END_IF;

	END_FOR;

	IF Loc.PowerStatus THEN
		gHMI.Widget.PowerGroup.Power.Style := 'Command';
	ELSE
		gHMI.Widget.PowerGroup.Power.Style := 'default';
	END_IF;

	//======================================
	//		  Vacuum Grubu Butonlarý
	//======================================

	IF gIO.In.Sealing.X2VacuumOK THEN
		gHMI.Widget.Button.HoldGlass.Style:= 'Command';
	ELSE
		gHMI.Widget.Button.HoldGlass.Style := 'default';
	END_IF;

	//======================================
	//		  Otomatikten manuel moda geçis
	//======================================
	IF ((gPML[PML_TASK_SEALING].SubStateCurrent = SUBS_WAIT_CMD OR gPML[PML_TASK_SEALING].StateCurrent = mpPACKML_STATE_IDLE) AND gPML[0].ModeID = PML_MODE_AUTO) OR ( gPML[0].ModeID = PML_MODE_MAN )THEN
		gHMI.Widget.PowerGroup.Manual.Enable := TRUE ;
	ELSE
		gHMI.Widget.PowerGroup.Manual.Enable := FALSE ;
	END_IF;

	//======================================
	//		  Ekran hareketleri
	//======================================
	IF gHMI.Status.EdgeBaseChange THEN
		gRecData.Speed.EdgeBase[1] := gRecData.Speed.EdgeBase[0];
		gRecData.Speed.EdgeBase[2] := gRecData.Speed.EdgeBase[0];
		gRecData.Speed.EdgeBase[3] := gRecData.Speed.EdgeBase[0];
		gHMI.Status.EdgeBaseChange := FALSE;
	END_IF;

	IF gHMI.Status.CompCloseChange THEN
		gRecData.Distance[gFixData.Config.SpacerType].CompClose[1] := 	gRecData.Distance[gFixData.Config.SpacerType].CompClose[0];
		gRecData.Distance[gFixData.Config.SpacerType].CompClose[2] := 	gRecData.Distance[gFixData.Config.SpacerType].CompClose[0];
		gRecData.Distance[gFixData.Config.SpacerType].CompClose[3] := 	gRecData.Distance[gFixData.Config.SpacerType].CompClose[0];
		gHMI.Status.CompCloseChange := FALSE;
	END_IF;

	IF gHMI.Status.CornerFillingChange THEN
		gRecData.Time[gFixData.Config.SpacerType].CornerFilling[1]	:= gRecData.Time[gFixData.Config.SpacerType].CornerFilling[0];
		gRecData.Time[gFixData.Config.SpacerType].CornerFilling[2]	:= gRecData.Time[gFixData.Config.SpacerType].CornerFilling[0];
		gRecData.Time[gFixData.Config.SpacerType].CornerFilling[3]	:= gRecData.Time[gFixData.Config.SpacerType].CornerFilling[0];
		gHMI.Status.CornerFillingChange	:= FALSE;
	END_IF;

	IF gHMI.Status.PreOpenChange THEN
		gRecData.Time[gFixData.Config.SpacerType].CompPreOpen[1]		:= gRecData.Time[gFixData.Config.SpacerType].CompPreOpen[0];
		gRecData.Time[gFixData.Config.SpacerType].CompPreOpen[2]		:= gRecData.Time[gFixData.Config.SpacerType].CompPreOpen[0];
		gRecData.Time[gFixData.Config.SpacerType].CompPreOpen[3]		:= gRecData.Time[gFixData.Config.SpacerType].CompPreOpen[0];
		gHMI.Status.PreOpenChange			:=FALSE;
	END_IF;

	IF gHMI.Status.StartPosChange THEN
		gRecData.Distance[gFixData.Config.SpacerType].StartUpComponent[1]	:=gRecData.Distance[gFixData.Config.SpacerType].StartUpComponent[0];
		gRecData.Distance[gFixData.Config.SpacerType].StartUpComponent[2]	:=gRecData.Distance[gFixData.Config.SpacerType].StartUpComponent[0];
		gRecData.Distance[gFixData.Config.SpacerType].StartUpComponent[3]	:=gRecData.Distance[gFixData.Config.SpacerType].StartUpComponent[0];
		gHMI.Status.StartPosChange			:=FALSE;
	END_IF;

	IF EDGEPOS(gRecData.Time[gFixData.Config.SpacerType].CompPreOpen[0] <> 0) THEN
		gRecData.Distance[gFixData.Config.SpacerType].StartUpComponent[0] := 0;
	END_IF;

	IF EDGEPOS(gRecData.Time[gFixData.Config.SpacerType].CompPreOpen[1] <> 0) THEN
		gRecData.Distance[gFixData.Config.SpacerType].StartUpComponent[1] := 0;
	END_IF;

	IF EDGEPOS(gRecData.Time[gFixData.Config.SpacerType].CompPreOpen[2] <> 0) THEN
		gRecData.Distance[gFixData.Config.SpacerType].StartUpComponent[2] := 0;
	END_IF;

	IF EDGEPOS(gRecData.Time[gFixData.Config.SpacerType].CompPreOpen[3] <> 0) THEN
		gRecData.Distance[gFixData.Config.SpacerType].StartUpComponent[3] := 0;
	END_IF;

	IF EDGEPOS(gRecData.Distance[gFixData.Config.SpacerType].StartUpComponent[0] <> 0) THEN
		gRecData.Time[gFixData.Config.SpacerType].CompPreOpen[0] := 0;
	END_IF;

	IF EDGEPOS(gRecData.Distance[gFixData.Config.SpacerType].StartUpComponent[1] <> 0) THEN
		gRecData.Time[gFixData.Config.SpacerType].CompPreOpen[1] := 0;
	END_IF;

	IF EDGEPOS(gRecData.Distance[gFixData.Config.SpacerType].StartUpComponent[2] <> 0) THEN
		gRecData.Time[gFixData.Config.SpacerType].CompPreOpen[2] := 0;
	END_IF;

	IF EDGEPOS(gRecData.Distance[gFixData.Config.SpacerType].StartUpComponent[3] <> 0) THEN
		gRecData.Time[gFixData.Config.SpacerType].CompPreOpen[3] := 0;
	END_IF;

	//======================================
	//		  Üretim Sayilarini resetleme.
	//======================================
	IF gHMI.Cmd.ProductionReset THEN
		gFixData.Production.Daily.DoubleGlass 	:= 0;
		gFixData.Production.Daily.TripleGlass 	:= 0;
		gFixData.Production.DailyMeterSqr		:= 0;
		gHMI.Cmd.ProductionReset := FALSE ;
	END_IF;
	IF gFixData.Production.oldDay <> DTStructure_0.day AND DTStructure_0.day <> 0 THEN
		gFixData.Production.Daily.DoubleGlass 	:= 0;
		gFixData.Production.Daily.TripleGlass 	:= 0;
		gFixData.Production.DailyMeterSqr		:= 0;
		gFixData.Production.oldDay				:= DTStructure_0.day;
	END_IF;

	IF gFixData.Production.oldMonth <> DTStructure_0.month  AND DTStructure_0.month <> 0 THEN
		gFixData.Production.Month.DoubleGlass 	:= 0;
		gFixData.Production.Month.TripleGlass 	:= 0;
		gFixData.Production.oldMonth 			:= DTStructure_0.month;
	END_IF;

	//======================================
	//		  Derinlik Tanimlama
	//======================================

	IF gHMI.Cmd.SetMaxDepthDigit THEN
		gHMI.Cmd.SetMaxDepthDigit := FALSE;
		gFixData.Depth.MasterDepthDigit := gIO.In.Sealing.aiDeepnesSignal ;
	END_IF;

	IF gHMI.Cmd.SetGlassSurfaceDepthDigit THEN
		gHMI.Cmd.SetGlassSurfaceDepthDigit := FALSE;
		gFixData.Depth.GlassSurfaceDigit := gIO.In.Sealing.aiDeepnesSignal ;
	END_IF;
END_ACTION
```

#### IOcontrolPage.st
```iecst
(*********************************************************************************
 * Copyright:
 * Author:    baranc
 * Created:   October 6, 2025/1:24 PM
 *********************************************************************************)
ACTION IOcontrolPage:

	//---------------------------
	// Seçilen kart için dogru kanal sayisini ve adlarini göster
	FOR i := 0 TO 15 DO
		IF ((IO_START_INDEX_SELECTED_SLOT[gHMI.IO_Control.SelectedSlot] + i) <=
			(IO_START_INDEX_SELECTED_SLOT[gHMI.IO_Control.SelectedSlot] + gHMI.IO_Control.MaxDpIndex) ) THEN  // check if the index corresponds to an empty IO channel
			gHMI.IO_Control.NameSelector[i]    := IO_START_INDEX_SELECTED_SLOT[gHMI.IO_Control.SelectedSlot] + i;
			gHMI.IO_Control.DatafieldStatus[i] := TRUE;
		ELSE
			gHMI.IO_Control.NameSelector[i]    := 32767;   // Nothing is mapped to the IO channel
			gHMI.IO_Control.DatafieldStatus[i] := FALSE; // buraya sayfayi gizlemek için erisicez
		END_IF
	END_FOR

	//---------------------------
	// Kartlar dijital ise maximum 1 degeri girilsin, Analog ise 32767
	IF (gHMI.IO_Control.TypeOfIO = DI_IO OR gHMI.IO_Control.TypeOfIO = DO_IO) THEN	// Limits for DI, DO
		gHMI.IO_Control.MaxForceValueLimit 	:= 0;
		gHMI.IO_Control.MaxForceValueLimit	:= 1;
	ELSE	// Limits for AI, AO
		gHMI.IO_Control.MinForceValueLimit 	:= 0;
		gHMI.IO_Control.MaxForceValueLimit	:= 32767;
	END_IF;

	//----------------------------------------------
	// Seçili kartin degistigini anlamak için
	gHMI.IO_Control.SelectedSlotOld  := gHMI.IO_Control.SelectedSlot;

END_ACTION
```

#### MachineLockPage.st
```iecst
(*********************************************************************************
 * Copyright:
 * Author:    baranc
 * Created:   October 8, 2025/9:10 AM
 *********************************************************************************)

ACTION MachineLockPage:
	//======================================
	//		Get Time
	//======================================

	DTStructureGetTime_0.enable := TRUE;
	DTStructureGetTime_0.pDTStructure := ADR(DTStructure_0);
	DTStructureGetTime_0();
	//Sistem zamanini çekelim.
	DTGetTime_0.enable 	:= TRUE;
	SystemTime			:= DTGetTime_0.DT1 ;
	DTGetTime_0();
	//SuperPassword hesaplama
	SuperPassword:= '';
	tempMonth	:= USINT_TO_STRING(DTStructure_0.month * 2);
	tempDay	:= USINT_TO_STRING(DTStructure_0.day * 2);
	brsstrcat(ADR(SuperPassword),ADR(tempDay));
	brsstrcat(ADR(SuperPassword),ADR(tempMonth));

	//Normal Password Hesaplama
	NormalPassword:= '';
	tempMonth	:= USINT_TO_STRING(DTStructure_0.month + 1);
	tempDay		:= USINT_TO_STRING(DTStructure_0.day + 1) ;
	brsstrcat(ADR(NormalPassword),ADR(tempDay));
	brsstrcat(ADR(NormalPassword),ADR(tempMonth));

	//Süper Sifre ile giris yapilirsa tamamen kapatilsin.
	IF gHMI.MachineLock.Login AND gHMI.MachineLock.Password = SuperPassword AND gHMI.UserName <> 'admin'  THEN
		gHMI.MachineLock.Enable		:= FALSE;
		gHMI.MachineLock.Password		:= '' ;
	END_IF;

	//Süper Sifre ile giris yapilirsa ve admin modundaysan tarih ayarlanabilir olacak.
	IF gHMI.MachineLock.Login AND gHMI.MachineLock.Password = SuperPassword AND gHMI.UserName = 'admin' THEN
		gHMI.Widget.MachineLock.Visible := TRUE;
		gHMI.MachineLock.Password		:= '' ;
	END_IF;

	//Sifre 2 ile giris yapilirsa mevcut süre 1 ay uzatilsin.
	IF gHMI.MachineLock.Login AND gHMI.MachineLock.Password = NormalPassword AND gHMI.MachineLock.oldDay <> DTStructure_0.day AND DTStructure_0.day <> 0 THEN
		gHMI.MachineLock.EndTime :=  gHMI.MachineLock.EndTime + t#14d + t#14d + t#2d;
		gHMI.MachineLock.Login		 := FALSE;
		gHMI.MachineLock.Password		:= '' ;
		gHMI.MachineLock.oldDay := DTStructure_0.day;
	END_IF;

	// eger kilitleme zamani geçmis ve makine kilitleme opsiyonu açiksa .
	IF (gHMI.MachineLock.EndTime < SystemTime) AND gHMI.MachineLock.Enable THEN
		gHMI.MachineLock.Lock := TRUE;
	ELSE
		gHMI.MachineLock.Lock := FALSE;
	END_IF;

	TON_Logout.IN := gHMI.Widget.MachineLock.Visible ;
	TON_Logout.PT := T#1m;

	IF TON_Logout.Q THEN
	  gHMI.Widget.MachineLock.Visible := FALSE;
	END_IF;

	TON_Logout();

END_ACTION
```
